LIN {X 0,Y 354.85,Z 275.906,A -85,B 0,C 180,E1 -13291.619,E2 -13291.619} C_VEL
LIN {X 0,Y 354.902,Z 275.901,A -85,B 0,C 180,E1 -13294.172,E2 -13294.172} C_VEL
LIN {X 0,Y 354.819,Z 275.911,A -85,B 0,C 180,E1 -13297.893,E2 -13297.893} C_VEL
LIN {X 0,Y 354.926,Z 275.898,A -85,B 0,C 180,E1 -13301.891,E2 -13301.891} C_VEL
LIN {X 0,Y 354.947,Z 275.897,A -85,B 0,C 180,E1 -13305.981,E2 -13305.981} C_VEL
LIN {X 0,Y 354.96,Z 275.894,A -85,B 0,C 180,E1 -13309.735,E2 -13309.735} C_VEL
LIN {X 0,Y 355.092,Z 275.876,A -85,B 0,C 180,E1 -13313.18,E2 -13313.18} C_VEL
LIN {X 0,Y 355.245,Z 275.86,A -85,B 0,C 180,E1 -13317.732,E2 -13317.732} C_VEL
LIN {X 0,Y 355.335,Z 275.85,A -85,B 0,C 180,E1 -13320,E2 -13320} C_VEL
LIN {X 0,Y 355.247,Z 275.86,A -85,B 0,C 180,E1 -13322.267,E2 -13322.267} C_VEL
LIN {X 0,Y 355.094,Z 275.875,A -85,B 0,C 180,E1 -13326.82,E2 -13326.82} C_VEL
LIN {X 0,Y 354.959,Z 275.894,A -85,B 0,C 180,E1 -13330.264,E2 -13330.264} C_VEL
LIN {X 0,Y 354.946,Z 275.896,A -85,B 0,C 180,E1 -13334.019,E2 -13334.019} C_VEL
LIN {X 0,Y 354.925,Z 275.898,A -85,B 0,C 180,E1 -13338.108,E2 -13338.108} C_VEL
LIN {X 0,Y 354.838,Z 275.908,A -85,B 0,C 180,E1 -13342.106,E2 -13342.106} C_VEL
LIN {X 0,Y 354.818,Z 275.914,A -85,B 0,C 180,E1 -13345.834,E2 -13345.834} C_VEL
LIN {X 0,Y 354.801,Z 275.915,A -85,B 0,C 180,E1 -13349.683,E2 -13349.683} C_VEL
LIN {X 0,Y 354.839,Z 276.09,A -85,B 0,C 180,E1 -13353.341,E2 -13353.341} C_VEL
LIN {X 0,Y 355.541,Z 279.989,A -85,B 0,C 180,E1 -13356.371,E2 -13356.371} C_VEL
LIN {X 0,Y 356.339,Z 284.55,A -85,B 0,C 180,E1 -13359.718,E2 -13359.718} C_VEL
LIN {X 0,Y 357.294,Z 289.71,A -85,B 0,C 180,E1 -13363.298,E2 -13363.298} C_VEL
LIN {X 0,Y 358.168,Z 294.793,A -85,B 0,C 180,E1 -13366.624,E2 -13366.624} C_VEL
LIN {X 0,Y 358.136,Z 298.563,A -85,B 0,C 180,E1 -13368.921,E2 -13368.921} C_VEL
LIN {X 0,Y 357.403,Z 304.661,A -85,B 0,C 180,E1 -13372.44,E2 -13372.44} C_VEL
LIN {X 0,Y 356.642,Z 310.823,A -85,B 0,C 180,E1 -13375.858,E2 -13375.858} C_VEL
LIN {X 0,Y 356.03,Z 316.866,A -85,B 0,C 180,E1 -13379.12,E2 -13379.12} C_VEL
LIN {X 0,Y 355.687,Z 320.46,A -85,B 0,C 180,E1 -13381.016,E2 -13381.016} C_VEL
LIN {X 0,Y 360.379,Z 339.057,A -85,B 0,C 180,E1 -13382.073,E2 -13382.073} C_VEL
LIN {X 0,Y 364.004,Z 355.046,A -85,B 0,C 180,E1 -13383.174,E2 -13383.174} C_VEL
LIN {X 0,Y 366.56,Z 369.171,A -85,B 0,C 180,E1 -13384.306,E2 -13384.306} C_VEL
LIN {X 0,Y 365.083,Z 383.132,A -85,B 0,C 180,E1 -13385.399,E2 -13385.399} C_VEL
LIN {X 0,Y 363.151,Z 396.131,A -85,B 0,C 180,E1 -13386.626,E2 -13386.626} C_VEL
LIN {X 0,Y 361.269,Z 409.429,A -85,B 0,C 180,E1 -13388.158,E2 -13388.158} C_VEL
LIN {X 0,Y 359.427,Z 421.341,A -85,B 0,C 180,E1 -13389.811,E2 -13389.811} C_VEL
LIN {X 0,Y 357.811,Z 432.557,A -85,B 0,C 180,E1 -13391.683,E2 -13391.683} C_VEL
LIN {X 0,Y 356.322,Z 442.487,A -85,B 0,C 180,E1 -13393.676,E2 -13393.676} C_VEL
LIN {X 0,Y 355.142,Z 451.425,A -85,B 0,C 180,E1 -13395.853,E2 -13395.853} C_VEL
LIN {X 0,Y 354.348,Z 458.565,A -85,B 0,C 180,E1 -13397.98,E2 -13397.98} C_VEL
LIN {X 0,Y 353.731,Z 464.736,A -85,B 0,C 180,E1 -13400.277,E2 -13400.277} C_VEL
LIN {X 0,Y 353.438,Z 469.47,A -85,B 0,C 180,E1 -13402.574,E2 -13402.574} C_VEL
LIN {X 0,Y 353.328,Z 472.143,A -85,B 0,C 180,E1 -13404.292,E2 -13404.292} C_VEL
LIN {X 0,Y 353.244,Z 474.612,A -85,B 0,C 180,E1 -13406.578,E2 -13406.578} C_VEL
LIN {X 0,Y 353.391,Z 475.823,A -85,B 0,C 180,E1 -13408.86,E2 -13408.86} C_VEL
LIN {X 0,Y 353.375,Z 475.789,A -85,B 0,C 180,E1 -13411.14,E2 -13411.14} C_VEL
LIN {X 0,Y 353.255,Z 474.542,A -85,B 0,C 180,E1 -13413.422,E2 -13413.422} C_VEL
LIN {X 0,Y 353.341,Z 472.092,A -85,B 0,C 180,E1 -13415.708,E2 -13415.708} C_VEL
LIN {X 0,Y 353.507,Z 468.395,A -85,B 0,C 180,E1 -13418,E2 -13418} C_VEL
LIN {X 0,Y 353.816,Z 463.389,A -85,B 0,C 180,E1 -13420.298,E2 -13420.298} C_VEL
LIN {X 0,Y 354.518,Z 456.97,A -85,B 0,C 180,E1 -13422.595,E2 -13422.595} C_VEL
LIN {X 0,Y 355.527,Z 449.023,A -85,B 0,C 180,E1 -13424.891,E2 -13424.891} C_VEL
LIN {X 0,Y 356.96,Z 439.375,A -85,B 0,C 180,E1 -13427.177,E2 -13427.177} C_VEL
LIN {X 0,Y 358.613,Z 429.339,A -85,B 0,C 180,E1 -13429.163,E2 -13429.163} C_VEL
LIN {X 0,Y 360.3,Z 419.297,A -85,B 0,C 180,E1 -13430.854,E2 -13430.854} C_VEL
LIN {X 0,Y 362.734,Z 405.658,A -85,B 0,C 180,E1 -13432.799,E2 -13432.799} C_VEL
LIN {X 0,Y 365.271,Z 391.753,A -85,B 0,C 180,E1 -13434.436,E2 -13434.436} C_VEL
LIN {X 0,Y 367.862,Z 377.541,A -85,B 0,C 180,E1 -13435.822,E2 -13435.822} C_VEL
LIN {X 0,Y 368.776,Z 371.059,A -85,B 0,C 180,E1 -13436.401,E2 -13436.401} C_VEL
LIN {X 0,Y 367.343,Z 351.718,A -85,B 0,C 180,E1 -13438.35,E2 -13438.35} C_VEL
LIN {X 0,Y 365.877,Z 341.967,A -85,B 0,C 180,E1 -13439.357,E2 -13439.357} C_VEL
LIN {X 0,Y 363.489,Z 331.98,A -85,B 0,C 180,E1 -13440.491,E2 -13440.491} C_VEL
LIN {X 0,Y 360.327,Z 322.118,A -85,B 0,C 180,E1 -13441.778,E2 -13441.778} C_VEL
LIN {X 0,Y 358.806,Z 317.901,A -85,B 0,C 180,E1 -13442.393,E2 -13442.393} C_VEL
LIN {X 0,Y 356.659,Z 312.833,A -85,B 0,C 180,E1 -13443.248,E2 -13443.248} C_VEL
LIN {X 0,Y 356.363,Z 310.972,A -85,B 0,C 180,E1 -13443.518,E2 -13443.518} C_VEL
LIN {X 0,Y 357.047,Z 306.93,A -85,B 0,C 180,E1 -13446.194,E2 -13446.194} C_VEL
LIN {X 0,Y 357.722,Z 303.241,A -85,B 0,C 180,E1 -13448.954,E2 -13448.954} C_VEL
LIN {X 0,Y 358.386,Z 299.982,A -85,B 0,C 180,E1 -13451.825,E2 -13451.825} C_VEL
LIN {X 0,Y 358.515,Z 298.431,A -85,B 0,C 180,E1 -13453.505,E2 -13453.505} C_VEL
LIN {X 0,Y 358.44,Z 297.199,A -85,B 0,C 180,E1 -13455.101,E2 -13455.101} C_VEL
LIN {X 0,Y 358.232,Z 296.25,A -85,B 0,C 180,E1 -13456.635,E2 -13456.635} C_VEL
LIN {X 0,Y 357.483,Z 294.847,A -85,B 0,C 180,E1 -13460.061,E2 -13460.061} C_VEL
LIN {X 0,Y 356.838,Z 294.398,A -85,B 0,C 180,E1 -13463.108,E2 -13463.108} C_VEL
LIN {X 0,Y 357.907,Z 296.935,A -85,B 0,C 180,E1 -13463.62,E2 -13463.62} C_VEL
LIN {X 0,Y 360.271,Z 300.003,A -85,B 0,C 180,E1 -13464.475,E2 -13464.475} C_VEL
LIN {X 0,Y 364.618,Z 306.868,A -85,B 0,C 180,E1 -13465.979,E2 -13465.979} C_VEL
LIN {X 0,Y 369.433,Z 316.686,A -85,B 0,C 180,E1 -13467.686,E2 -13467.686} C_VEL
LIN {X 0,Y 372.523,Z 325.556,A -85,B 0,C 180,E1 -13468.961,E2 -13468.961} C_VEL
LIN {X 0,Y 372.708,Z 327.732,A -85,B 0,C 180,E1 -13469.187,E2 -13469.187} C_VEL
LIN {X 0,Y 370.521,Z 341.272,A -85,B 0,C 180,E1 -13470.296,E2 -13470.296} C_VEL
LIN {X 0,Y 368.081,Z 355.561,A -85,B 0,C 180,E1 -13471.706,E2 -13471.706} C_VEL
LIN {X 0,Y 365.485,Z 369.993,A -85,B 0,C 180,E1 -13473.444,E2 -13473.444} C_VEL
LIN {X 0,Y 363.155,Z 382.14,A -85,B 0,C 180,E1 -13475.211,E2 -13475.211} C_VEL
LIN {X 0,Y 361.133,Z 392.946,A -85,B 0,C 180,E1 -13477.094,E2 -13477.094} C_VEL
LIN {X 0,Y 358.991,Z 403.616,A -85,B 0,C 180,E1 -13479.367,E2 -13479.367} C_VEL
LIN {X 0,Y 357.704,Z 410.335,A -85,B 0,C 180,E1 -13481.084,E2 -13481.084} C_VEL
LIN {X 0,Y 356.334,Z 417.681,A -85,B 0,C 180,E1 -13483.383,E2 -13483.383} C_VEL
LIN {X 0,Y 355.285,Z 423.605,A -85,B 0,C 180,E1 -13485.764,E2 -13485.764} C_VEL
LIN {X 0,Y 354.732,Z 426.779,A -85,B 0,C 180,E1 -13487.413,E2 -13487.413} C_VEL
LIN {X 0,Y 354.107,Z 430.099,A -85,B 0,C 180,E1 -13489.711,E2 -13489.711} C_VEL
LIN {X 0,Y 353.786,Z 432.114,A -85,B 0,C 180,E1 -13492.007,E2 -13492.007} C_VEL
LIN {X 0,Y 353.631,Z 432.891,A -85,B 0,C 180,E1 -13494.297,E2 -13494.297} C_VEL
LIN {X 0,Y 353.541,Z 432.443,A -85,B 0,C 180,E1 -13496.581,E2 -13496.581} C_VEL
LIN {X 0,Y 353.533,Z 430.76,A -85,B 0,C 180,E1 -13498.861,E2 -13498.861} C_VEL
LIN {X 0,Y 353.572,Z 427.813,A -85,B 0,C 180,E1 -13501.139,E2 -13501.139} C_VEL
LIN {X 0,Y 353.949,Z 423.542,A -85,B 0,C 180,E1 -13503.415,E2 -13503.415} C_VEL
LIN {X 0,Y 354.362,Z 419.416,A -85,B 0,C 180,E1 -13505.121,E2 -13505.121} C_VEL
LIN {X 0,Y 354.772,Z 412.637,A -85,B 0,C 180,E1 -13507.398,E2 -13507.398} C_VEL
LIN {X 0,Y 355.642,Z 404.164,A -85,B 0,C 180,E1 -13509.67,E2 -13509.67} C_VEL
LIN {X 0,Y 356.697,Z 395.156,A -85,B 0,C 180,E1 -13511.652,E2 -13511.652} C_VEL
LIN {X 0,Y 357.892,Z 384.378,A -85,B 0,C 180,E1 -13513.63,E2 -13513.63} C_VEL
LIN {X 0,Y 359.228,Z 373.388,A -85,B 0,C 180,E1 -13515.315,E2 -13515.315} C_VEL
LIN {X 0,Y 360.681,Z 360.339,A -85,B 0,C 180,E1 -13516.995,E2 -13516.995} C_VEL
LIN {X 0,Y 362.03,Z 347.331,A -85,B 0,C 180,E1 -13518.389,E2 -13518.389} C_VEL
LIN {X 0,Y 363.53,Z 333.259,A -85,B 0,C 180,E1 -13519.628,E2 -13519.628} C_VEL
LIN {X 0,Y 364.782,Z 317.486,A -85,B 0,C 180,E1 -13520.757,E2 -13520.757} C_VEL
LIN {X 0,Y 360.614,Z 301.762,A -85,B 0,C 180,E1 -13521.924,E2 -13521.924} C_VEL
LIN {X 0,Y 355.886,Z 285.872,A -85,B 0,C 180,E1 -13522.918,E2 -13522.918} C_VEL
LIN {X 0,Y 353.92,Z 279.21,A -85,B 0,C 180,E1 -13523.289,E2 -13523.289} C_VEL
LIN {X 0,Y 353.968,Z 276.176,A -85,B 0,C 180,E1 -13526.687,E2 -13526.687} C_VEL
LIN {X 0,Y 354.293,Z 275.978,A -85,B 0,C 180,E1 -13529.731,E2 -13529.731} C_VEL
LIN {X 0,Y 354.529,Z 275.947,A -85,B 0,C 180,E1 -13532.36,E2 -13532.36} C_VEL
LIN {X 0,Y 354.794,Z 275.914,A -85,B 0,C 180,E1 -13535.692,E2 -13535.692} C_VEL
LIN {X 0,Y 354.827,Z 275.912,A -85,B 0,C 180,E1 -13539.424,E2 -13539.424} C_VEL
LIN {X 0,Y 354.791,Z 275.918,A -85,B 0,C 180,E1 -13542.867,E2 -13542.867} C_VEL
LIN {X 0,Y 354.77,Z 275.916,A -85,B 0,C 180,E1 -13546.104,E2 -13546.104} C_VEL
LIN {X 0,Y 354.791,Z 275.916,A -85,B 0,C 180,E1 -13549.179,E2 -13549.179} C_VEL
LIN {X 0,Y 354.81,Z 275.913,A -85,B 0,C 180,E1 -13552.403,E2 -13552.403} C_VEL
LIN {X 0,Y 354.815,Z 275.914,A -85,B 0,C 180,E1 -13554.941,E2 -13554.941} C_VEL
LIN {X 0,Y 354.796,Z 275.916,A -85,B 0,C 180,E1 -13558.405,E2 -13558.405} C_VEL
LIN {X 0,Y 354.849,Z 275.906,A -85,B 0,C 180,E1 -13561.619,E2 -13561.619} C_VEL
LIN {X 0,Y 354.901,Z 275.902,A -85,B 0,C 180,E1 -13564.173,E2 -13564.173} C_VEL
LIN {X 0,Y 354.811,Z 275.912,A -85,B 0,C 180,E1 -13567.892,E2 -13567.892} C_VEL
LIN {X 0,Y 354.925,Z 275.898,A -85,B 0,C 180,E1 -13571.892,E2 -13571.892} C_VEL
LIN {X 0,Y 354.946,Z 275.897,A -85,B 0,C 180,E1 -13575.981,E2 -13575.981} C_VEL
LIN {X 0,Y 354.981,Z 275.891,A -85,B 0,C 180,E1 -13579.736,E2 -13579.736} C_VEL
LIN {X 0,Y 355.091,Z 275.876,A -85,B 0,C 180,E1 -13583.18,E2 -13583.18} C_VEL
LIN {X 0,Y 355.238,Z 275.861,A -85,B 0,C 180,E1 -13587.732,E2 -13587.732} C_VEL
LIN {X 0,Y 355.355,Z 275.848,A -85,B 0,C 180,E1 -13590,E2 -13590} C_VEL
LIN {X 0,Y 355.244,Z 275.859,A -85,B 0,C 180,E1 -13592.268,E2 -13592.268} C_VEL
LIN {X 0,Y 355.102,Z 275.875,A -85,B 0,C 180,E1 -13596.82,E2 -13596.82} C_VEL
LIN {X 0,Y 354.959,Z 275.894,A -85,B 0,C 180,E1 -13600.265,E2 -13600.265} C_VEL
LIN {X 0,Y 354.946,Z 275.896,A -85,B 0,C 180,E1 -13604.019,E2 -13604.019} C_VEL
LIN {X 0,Y 354.926,Z 275.898,A -85,B 0,C 180,E1 -13608.108,E2 -13608.108} C_VEL
LIN {X 0,Y 354.838,Z 275.908,A -85,B 0,C 180,E1 -13612.106,E2 -13612.106} C_VEL
LIN {X 0,Y 354.903,Z 275.902,A -85,B 0,C 180,E1 -13615.827,E2 -13615.827} C_VEL
LIN {X 0,Y 354.821,Z 275.912,A -85,B 0,C 180,E1 -13619.682,E2 -13619.682} C_VEL
LIN {X 0,Y 354.809,Z 275.913,A -85,B 0,C 180,E1 -13623.702,E2 -13623.702} C_VEL
LIN {X 0,Y 354.799,Z 275.912,A -85,B 0,C 180,E1 -13626.46,E2 -13626.46} C_VEL
LIN {X 0,Y 354.771,Z 275.919,A -85,B 0,C 180,E1 -13629.412,E2 -13629.412} C_VEL
LIN {X 0,Y 354.787,Z 275.918,A -85,B 0,C 180,E1 -13632.866,E2 -13632.866} C_VEL
LIN {X 0,Y 354.769,Z 275.916,A -85,B 0,C 180,E1 -13636.104,E2 -13636.104} C_VEL
LIN {X 0,Y 354.785,Z 275.917,A -85,B 0,C 180,E1 -13638.708,E2 -13638.708} C_VEL
LIN {X 0,Y 354.146,Z 276.003,A -85,B 0,C 180,E1 -13639.657,E2 -13639.657} C_VEL
LIN {X 0,Y 351.276,Z 276.358,A -85,B 0,C 180,E1 -13641.199,E2 -13641.199} C_VEL
LIN {X 0,Y 348.845,Z 276.656,A -85,B 0,C 180,E1 -13642.447,E2 -13642.447} C_VEL
LIN {X 0,Y 347.829,Z 276.781,A -85,B 0,C 180,E1 -13643.413,E2 -13643.413} C_VEL
LIN {X 0,Y 347.762,Z 276.788,A -85,B 0,C 180,E1 -13643.741,E2 -13643.741} C_VEL
LIN {X 0,Y 347.737,Z 276.796,A -85,B 0,C 180,E1 -13646.928,E2 -13646.928} C_VEL
LIN {X 0,Y 347.782,Z 276.789,A -85,B 0,C 180,E1 -13650.988,E2 -13650.988} C_VEL
LIN {X 0,Y 347.834,Z 276.779,A -85,B 0,C 180,E1 -13653.608,E2 -13653.608} C_VEL
LIN {X 0,Y 347.789,Z 276.788,A -85,B 0,C 180,E1 -13656.162,E2 -13656.162} C_VEL
LIN {X 0,Y 347.811,Z 276.784,A -85,B 0,C 180,E1 -13659.909,E2 -13659.909} C_VEL
LIN {X 0,Y 347.87,Z 276.78,A -85,B 0,C 180,E1 -13662.359,E2 -13662.359} C_VEL
LIN {X 0,Y 347.901,Z 276.774,A -85,B 0,C 180,E1 -13665.971,E2 -13665.971} C_VEL
LIN {X 0,Y 347.901,Z 276.772,A -85,B 0,C 180,E1 -13669.524,E2 -13669.524} C_VEL
LIN {X 0,Y 348.059,Z 276.752,A -85,B 0,C 180,E1 -13673.041,E2 -13673.041} C_VEL
LIN {X 0,Y 348.207,Z 276.736,A -85,B 0,C 180,E1 -13677.686,E2 -13677.686} C_VEL
LIN {X 0,Y 348.287,Z 276.728,A -85,B 0,C 180,E1 -13680,E2 -13680} C_VEL
LIN {X 0,Y 348.21,Z 276.736,A -85,B 0,C 180,E1 -13682.313,E2 -13682.313} C_VEL
LIN {X 0,Y 348.06,Z 276.751,A -85,B 0,C 180,E1 -13686.958,E2 -13686.958} C_VEL
LIN {X 0,Y 347.9,Z 276.772,A -85,B 0,C 180,E1 -13690.475,E2 -13690.475} C_VEL
LIN {X 0,Y 347.902,Z 276.773,A -85,B 0,C 180,E1 -13694.149,E2 -13694.149} C_VEL
LIN {X 0,Y 347.894,Z 276.773,A -85,B 0,C 180,E1 -13698.29,E2 -13698.29} C_VEL
LIN {X 0,Y 347.793,Z 276.789,A -85,B 0,C 180,E1 -13701.635,E2 -13701.635} C_VEL
LIN {X 0,Y 347.772,Z 276.79,A -85,B 0,C 180,E1 -13705.111,E2 -13705.111} C_VEL
LIN {X 0,Y 347.738,Z 276.794,A -85,B 0,C 180,E1 -13707.7,E2 -13707.7} C_VEL
LIN {X 0,Y 347.742,Z 276.794,A -85,B 0,C 180,E1 -13710.348,E2 -13710.348} C_VEL
LIN {X 0,Y 347.759,Z 276.839,A -85,B 0,C 180,E1 -13712.752,E2 -13712.752} C_VEL
LIN {X 0,Y 348.553,Z 281.23,A -85,B 0,C 180,E1 -13716.241,E2 -13716.241} C_VEL
LIN {X 0,Y 349.482,Z 286.512,A -85,B 0,C 180,E1 -13720.166,E2 -13720.166} C_VEL
LIN {X 0,Y 350.247,Z 290.566,A -85,B 0,C 180,E1 -13723.018,E2 -13723.018} C_VEL
LIN {X 0,Y 351.056,Z 295.188,A -85,B 0,C 180,E1 -13726.113,E2 -13726.113} C_VEL
LIN {X 0,Y 351.239,Z 297.774,A -85,B 0,C 180,E1 -13727.76,E2 -13727.76} C_VEL
LIN {X 0,Y 350.724,Z 302.912,A -85,B 0,C 180,E1 -13730.834,E2 -13730.834} C_VEL
LIN {X 0,Y 349.923,Z 309.065,A -85,B 0,C 180,E1 -13734.377,E2 -13734.377} C_VEL
LIN {X 0,Y 349.265,Z 315.014,A -85,B 0,C 180,E1 -13737.686,E2 -13737.686} C_VEL
LIN {X 0,Y 348.706,Z 320.201,A -85,B 0,C 180,E1 -13740.492,E2 -13740.492} C_VEL
LIN {X 0,Y 353.123,Z 337.808,A -85,B 0,C 180,E1 -13741.507,E2 -13741.507} C_VEL
LIN {X 0,Y 356.956,Z 354.401,A -85,B 0,C 180,E1 -13742.679,E2 -13742.679} C_VEL
LIN {X 0,Y 359.766,Z 370.145,A -85,B 0,C 180,E1 -13743.975,E2 -13743.975} C_VEL
LIN {X 0,Y 359.333,Z 375.801,A -85,B 0,C 180,E1 -13744.416,E2 -13744.416} C_VEL
LIN {X 0,Y 357.43,Z 389.485,A -85,B 0,C 180,E1 -13745.612,E2 -13745.612} C_VEL
LIN {X 0,Y 355.468,Z 402.63,A -85,B 0,C 180,E1 -13747.015,E2 -13747.015} C_VEL
LIN {X 0,Y 353.448,Z 415.792,A -85,B 0,C 180,E1 -13748.722,E2 -13748.722} C_VEL
LIN {X 0,Y 351.707,Z 426.828,A -85,B 0,C 180,E1 -13750.445,E2 -13750.445} C_VEL
LIN {X 0,Y 350.016,Z 437.641,A -85,B 0,C 180,E1 -13752.471,E2 -13752.471} C_VEL
LIN {X 0,Y 348.709,Z 446.678,A -85,B 0,C 180,E1 -13754.511,E2 -13754.511} C_VEL
LIN {X 0,Y 347.757,Z 454.196,A -85,B 0,C 180,E1 -13756.561,E2 -13756.561} C_VEL
LIN {X 0,Y 346.976,Z 461.209,A -85,B 0,C 180,E1 -13758.906,E2 -13758.906} C_VEL
LIN {X 0,Y 346.496,Z 466.696,A -85,B 0,C 180,E1 -13761.25,E2 -13761.25} C_VEL
LIN {X 0,Y 346.314,Z 469.901,A -85,B 0,C 180,E1 -13763.006,E2 -13763.006} C_VEL
LIN {X 0,Y 346.218,Z 473.045,A -85,B 0,C 180,E1 -13765.343,E2 -13765.343} C_VEL
LIN {X 0,Y 346.201,Z 474.903,A -85,B 0,C 180,E1 -13767.673,E2 -13767.673} C_VEL
LIN {X 0,Y 346.311,Z 475.366,A -85,B 0,C 180,E1 -13768.837,E2 -13768.837} C_VEL
LIN {X 0,Y 346.297,Z 475.367,A -85,B 0,C 180,E1 -13771.163,E2 -13771.163} C_VEL
LIN {X 0,Y 346.176,Z 474.151,A -85,B 0,C 180,E1 -13773.492,E2 -13773.492} C_VEL
LIN {X 0,Y 346.285,Z 471.458,A -85,B 0,C 180,E1 -13776.028,E2 -13776.028} C_VEL
LIN {X 0,Y 346.427,Z 468.077,A -85,B 0,C 180,E1 -13778.164,E2 -13778.164} C_VEL
LIN {X 0,Y 346.767,Z 463.108,A -85,B 0,C 180,E1 -13780.51,E2 -13780.51} C_VEL
LIN {X 0,Y 347.506,Z 456.739,A -85,B 0,C 180,E1 -13782.854,E2 -13782.854} C_VEL
LIN {X 0,Y 348.59,Z 448.878,A -85,B 0,C 180,E1 -13785.195,E2 -13785.195} C_VEL
LIN {X 0,Y 350.118,Z 439.372,A -85,B 0,C 180,E1 -13787.524,E2 -13787.524} C_VEL
LIN {X 0,Y 351.864,Z 429.469,A -85,B 0,C 180,E1 -13789.546,E2 -13789.546} C_VEL
LIN {X 0,Y 353.998,Z 417.872,A -85,B 0,C 180,E1 -13791.548,E2 -13791.548} C_VEL
LIN {X 0,Y 356.631,Z 404.158,A -85,B 0,C 180,E1 -13793.52,E2 -13793.52} C_VEL
LIN {X 0,Y 359.38,Z 390.278,A -85,B 0,C 180,E1 -13795.172,E2 -13795.172} C_VEL
LIN {X 0,Y 362.3,Z 375.244,A -85,B 0,C 180,E1 -13796.653,E2 -13796.653} C_VEL
LIN {X 0,Y 362.592,Z 372.475,A -85,B 0,C 180,E1 -13796.925,E2 -13796.925} C_VEL
LIN {X 0,Y 361.547,Z 353.176,A -85,B 0,C 180,E1 -13798.986,E2 -13798.986} C_VEL
LIN {X 0,Y 359.907,Z 342.138,A -85,B 0,C 180,E1 -13800.231,E2 -13800.231} C_VEL
LIN {X 0,Y 357.553,Z 332.291,A -85,B 0,C 180,E1 -13801.489,E2 -13801.489} C_VEL
LIN {X 0,Y 356.069,Z 327.128,A -85,B 0,C 180,E1 -13802.203,E2 -13802.203} C_VEL
LIN {X 0,Y 354.474,Z 322.345,A -85,B 0,C 180,E1 -13802.949,E2 -13802.949} C_VEL
LIN {X 0,Y 352.61,Z 317.64,A -85,B 0,C 180,E1 -13803.79,E2 -13803.79} C_VEL
LIN {X 0,Y 352.385,Z 316.525,A -85,B 0,C 180,E1 -13803.948,E2 -13803.948} C_VEL
LIN {X 0,Y 350.293,Z 311.942,A -85,B 0,C 180,E1 -13804.934,E2 -13804.934} C_VEL
LIN {X 0,Y 349.808,Z 309.463,A -85,B 0,C 180,E1 -13805.353,E2 -13805.353} C_VEL
LIN {X 0,Y 350.649,Z 305.114,A -85,B 0,C 180,E1 -13808.587,E2 -13808.587} C_VEL
LIN {X 0,Y 351.322,Z 302.003,A -85,B 0,C 180,E1 -13811.311,E2 -13811.311} C_VEL
LIN {X 0,Y 351.565,Z 299.578,A -85,B 0,C 180,E1 -13813.974,E2 -13813.974} C_VEL
LIN {X 0,Y 351.37,Z 298.141,A -85,B 0,C 180,E1 -13816.06,E2 -13816.06} C_VEL
LIN {X 0,Y 350.861,Z 296.886,A -85,B 0,C 180,E1 -13818.623,E2 -13818.623} C_VEL
LIN {X 0,Y 350.289,Z 296.173,A -85,B 0,C 180,E1 -13821.282,E2 -13821.282} C_VEL
LIN {X 0,Y 350.697,Z 297.494,A -85,B 0,C 180,E1 -13821.593,E2 -13821.593} C_VEL
LIN {X 0,Y 351.72,Z 299.107,A -85,B 0,C 180,E1 -13822.118,E2 -13822.118} C_VEL
LIN {X 0,Y 353.274,Z 300.437,A -85,B 0,C 180,E1 -13822.727,E2 -13822.727} C_VEL
LIN {X 0,Y 355.163,Z 303.662,A -85,B 0,C 180,E1 -13823.584,E2 -13823.584} C_VEL
LIN {X 0,Y 358.458,Z 308.693,A -85,B 0,C 180,E1 -13824.883,E2 -13824.883} C_VEL
LIN {X 0,Y 362.509,Z 316.531,A -85,B 0,C 180,E1 -13826.476,E2 -13826.476} C_VEL
LIN {X 0,Y 365.589,Z 324.049,A -85,B 0,C 180,E1 -13827.763,E2 -13827.763} C_VEL
LIN {X 0,Y 367.18,Z 329.285,A -85,B 0,C 180,E1 -13828.535,E2 -13828.535} C_VEL
LIN {X 0,Y 364.385,Z 345.126,A -85,B 0,C 180,E1 -13829.903,E2 -13829.903} C_VEL
LIN {X 0,Y 361.806,Z 358.925,A -85,B 0,C 180,E1 -13831.362,E2 -13831.362} C_VEL
LIN {X 0,Y 359.307,Z 371.574,A -85,B 0,C 180,E1 -13832.95,E2 -13832.95} C_VEL
LIN {X 0,Y 356.579,Z 384.833,A -85,B 0,C 180,E1 -13834.97,E2 -13834.97} C_VEL
LIN {X 0,Y 354.351,Z 395.455,A -85,B 0,C 180,E1 -13836.939,E2 -13836.939} C_VEL
LIN {X 0,Y 352.393,Z 404.582,A -85,B 0,C 180,E1 -13838.962,E2 -13838.962} C_VEL
LIN {X 0,Y 350.595,Z 413.15,A -85,B 0,C 180,E1 -13841.293,E2 -13841.293} C_VEL
LIN {X 0,Y 349.202,Z 420.004,A -85,B 0,C 180,E1 -13843.635,E2 -13843.635} C_VEL
LIN {X 0,Y 348.214,Z 425.335,A -85,B 0,C 180,E1 -13845.984,E2 -13845.984} C_VEL
LIN {X 0,Y 347.341,Z 429.262,A -85,B 0,C 180,E1 -13848.327,E2 -13848.327} C_VEL
LIN {X 0,Y 346.899,Z 431.859,A -85,B 0,C 180,E1 -13850.673,E2 -13850.673} C_VEL
LIN {X 0,Y 346.609,Z 433.214,A -85,B 0,C 180,E1 -13853.012,E2 -13853.012} C_VEL
LIN {X 0,Y 346.454,Z 433.33,A -85,B 0,C 180,E1 -13855.346,E2 -13855.346} C_VEL
LIN {X 0,Y 346.509,Z 432.212,A -85,B 0,C 180,E1 -13857.675,E2 -13857.675} C_VEL
LIN {X 0,Y 346.447,Z 429.864,A -85,B 0,C 180,E1 -13860,E2 -13860} C_VEL
LIN {X 0,Y 346.669,Z 426.21,A -85,B 0,C 180,E1 -13862.324,E2 -13862.324} C_VEL
LIN {X 0,Y 347.157,Z 421.199,A -85,B 0,C 180,E1 -13864.645,E2 -13864.645} C_VEL
LIN {X 0,Y 347.601,Z 414.75,A -85,B 0,C 180,E1 -13866.968,E2 -13866.968} C_VEL
LIN {X 0,Y 348.375,Z 406.661,A -85,B 0,C 180,E1 -13869.288,E2 -13869.288} C_VEL
LIN {X 0,Y 349.39,Z 398.055,A -85,B 0,C 180,E1 -13871.311,E2 -13871.311} C_VEL
LIN {X 0,Y 350.619,Z 387.75,A -85,B 0,C 180,E1 -13873.328,E2 -13873.328} C_VEL
LIN {X 0,Y 351.866,Z 377.299,A -85,B 0,C 180,E1 -13875.05,E2 -13875.05} C_VEL
LIN {X 0,Y 353.381,Z 364.902,A -85,B 0,C 180,E1 -13876.761,E2 -13876.761} C_VEL
LIN {X 0,Y 354.824,Z 351.082,A -85,B 0,C 180,E1 -13878.35,E2 -13878.35} C_VEL
LIN {X 0,Y 356.276,Z 337.965,A -85,B 0,C 180,E1 -13879.594,E2 -13879.594} C_VEL
LIN {X 0,Y 357.575,Z 323.561,A -85,B 0,C 180,E1 -13880.719,E2 -13880.719} C_VEL
LIN {X 0,Y 357.86,Z 318.505,A -85,B 0,C 180,E1 -13881.07,E2 -13881.07} C_VEL
LIN {X 0,Y 353.728,Z 302.534,A -85,B 0,C 180,E1 -13882.293,E2 -13882.293} C_VEL
LIN {X 0,Y 348.767,Z 286.075,A -85,B 0,C 180,E1 -13883.345,E2 -13883.345} C_VEL
LIN {X 0,Y 346.865,Z 279.6,A -85,B 0,C 180,E1 -13883.739,E2 -13883.739} C_VEL
LIN {X 0,Y 346.916,Z 276.901,A -85,B 0,C 180,E1 -13886.953,E2 -13886.953} C_VEL
LIN {X 0,Y 347.302,Z 276.846,A -85,B 0,C 180,E1 -13890.392,E2 -13890.392} C_VEL
LIN {X 0,Y 347.646,Z 276.803,A -85,B 0,C 180,E1 -13894.018,E2 -13894.018} C_VEL
LIN {X 0,Y 347.758,Z 276.793,A -85,B 0,C 180,E1 -13897.322,E2 -13897.322} C_VEL
LIN {X 0,Y 347.734,Z 276.793,A -85,B 0,C 180,E1 -13900.297,E2 -13900.297} C_VEL
LIN {X 0,Y 347.726,Z 276.795,A -85,B 0,C 180,E1 -13903.408,E2 -13903.408} C_VEL
LIN {X 0,Y 347.728,Z 276.797,A -85,B 0,C 180,E1 -13906.686,E2 -13906.686} C_VEL
LIN {X 0,Y 347.75,Z 276.791,A -85,B 0,C 180,E1 -13910.173,E2 -13910.173} C_VEL
LIN {X 0,Y 347.764,Z 276.793,A -85,B 0,C 180,E1 -13912.679,E2 -13912.679} C_VEL
LIN {X 0,Y 347.751,Z 276.79,A -85,B 0,C 180,E1 -13915.956,E2 -13915.956} C_VEL
LIN {X 0,Y 347.752,Z 276.79,A -85,B 0,C 180,E1 -13919.652,E2 -13919.652} C_VEL
LIN {X 0,Y 347.833,Z 276.78,A -85,B 0,C 180,E1 -13923.608,E2 -13923.608} C_VEL
LIN {X 0,Y 347.785,Z 276.789,A -85,B 0,C 180,E1 -13926.161,E2 -13926.161} C_VEL
LIN {X 0,Y 347.81,Z 276.784,A -85,B 0,C 180,E1 -13929.909,E2 -13929.909} C_VEL
LIN {X 0,Y 347.869,Z 276.78,A -85,B 0,C 180,E1 -13932.359,E2 -13932.359} C_VEL
LIN {X 0,Y 347.901,Z 276.775,A -85,B 0,C 180,E1 -13935.971,E2 -13935.971} C_VEL
LIN {X 0,Y 347.931,Z 276.768,A -85,B 0,C 180,E1 -13939.526,E2 -13939.526} C_VEL
LIN {X 0,Y 348.058,Z 276.752,A -85,B 0,C 180,E1 -13943.041,E2 -13943.041} C_VEL
LIN {X 0,Y 348.199,Z 276.737,A -85,B 0,C 180,E1 -13947.686,E2 -13947.686} C_VEL
LIN {X 0,Y 348.306,Z 276.726,A -85,B 0,C 180,E1 -13950,E2 -13950} C_VEL
LIN {X 0,Y 348.206,Z 276.735,A -85,B 0,C 180,E1 -13952.314,E2 -13952.314} C_VEL
LIN {X 0,Y 348.067,Z 276.751,A -85,B 0,C 180,E1 -13956.959,E2 -13956.959} C_VEL
LIN {X 0,Y 347.899,Z 276.772,A -85,B 0,C 180,E1 -13960.475,E2 -13960.475} C_VEL
LIN {X 0,Y 347.902,Z 276.773,A -85,B 0,C 180,E1 -13964.15,E2 -13964.15} C_VEL
LIN {X 0,Y 347.894,Z 276.773,A -85,B 0,C 180,E1 -13968.29,E2 -13968.29} C_VEL
LIN {X 0,Y 347.792,Z 276.789,A -85,B 0,C 180,E1 -13971.635,E2 -13971.635} C_VEL
LIN {X 0,Y 347.816,Z 276.785,A -85,B 0,C 180,E1 -13975.108,E2 -13975.108} C_VEL
LIN {X 0,Y 347.811,Z 276.785,A -85,B 0,C 180,E1 -13977.694,E2 -13977.694} C_VEL
LIN {X 0,Y 347.752,Z 276.79,A -85,B 0,C 180,E1 -13980.348,E2 -13980.348} C_VEL
LIN {X 0,Y 347.751,Z 276.79,A -85,B 0,C 180,E1 -13984.044,E2 -13984.044} C_VEL
LIN {X 0,Y 347.759,Z 276.793,A -85,B 0,C 180,E1 -13987.321,E2 -13987.321} C_VEL
LIN {X 0,Y 347.744,Z 276.792,A -85,B 0,C 180,E1 -13991.601,E2 -13991.601} C_VEL
LIN {X 0,Y 347.707,Z 276.8,A -85,B 0,C 180,E1 -13995.027,E2 -13995.027} C_VEL
LIN {X 0,Y 347.734,Z 276.791,A -85,B 0,C 180,E1 -13998.699,E2 -13998.699} C_VEL
LIN {X 0,Y 347.777,Z 276.787,A -85,B 0,C 180,E1 -14002.011,E2 -14002.011} C_VEL
LIN {X 0,Y 347.762,Z 276.788,A -85,B 0,C 180,E1 -14003.741,E2 -14003.741} C_VEL
LIN {X 0,Y 347.122,Z 276.873,A -85,B 0,C 180,E1 -14004.706,E2 -14004.706} C_VEL
LIN {X 0,Y 344.232,Z 277.23,A -85,B 0,C 180,E1 -14006.276,E2 -14006.276} C_VEL
LIN {X 0,Y 341.782,Z 277.533,A -85,B 0,C 180,E1 -14007.547,E2 -14007.547} C_VEL
LIN {X 0,Y 340.761,Z 277.665,A -85,B 0,C 180,E1 -14008.531,E2 -14008.531} C_VEL
LIN {X 0,Y 340.696,Z 277.671,A -85,B 0,C 180,E1 -14008.865,E2 -14008.865} C_VEL
LIN {X 0,Y 340.78,Z 277.663,A -85,B 0,C 180,E1 -14012.475,E2 -14012.475} C_VEL
LIN {X 0,Y 340.758,Z 277.661,A -85,B 0,C 180,E1 -14015.638,E2 -14015.638} C_VEL
LIN {X 0,Y 340.738,Z 277.663,A -85,B 0,C 180,E1 -14019.473,E2 -14019.473} C_VEL
LIN {X 0,Y 340.862,Z 277.65,A -85,B 0,C 180,E1 -14021.984,E2 -14021.984} C_VEL
LIN {X 0,Y 340.873,Z 277.648,A -85,B 0,C 180,E1 -14025.705,E2 -14025.705} C_VEL
LIN {X 0,Y 340.852,Z 277.649,A -85,B 0,C 180,E1 -14029.305,E2 -14029.305} C_VEL
LIN {X 0,Y 341.006,Z 277.63,A -85,B 0,C 180,E1 -14032.896,E2 -14032.896} C_VEL
LIN {X 0,Y 341.168,Z 277.612,A -85,B 0,C 180,E1 -14037.638,E2 -14037.638} C_VEL
LIN {X 0,Y 341.239,Z 277.606,A -85,B 0,C 180,E1 -14040,E2 -14040} C_VEL
LIN {X 0,Y 341.171,Z 277.612,A -85,B 0,C 180,E1 -14042.361,E2 -14042.361} C_VEL
LIN {X 0,Y 341.007,Z 277.63,A -85,B 0,C 180,E1 -14047.103,E2 -14047.103} C_VEL
LIN {X 0,Y 340.851,Z 277.649,A -85,B 0,C 180,E1 -14050.694,E2 -14050.694} C_VEL
LIN {X 0,Y 340.866,Z 277.648,A -85,B 0,C 180,E1 -14054.324,E2 -14054.324} C_VEL
LIN {X 0,Y 340.84,Z 277.651,A -85,B 0,C 180,E1 -14058.466,E2 -14058.466} C_VEL
LIN {X 0,Y 340.756,Z 277.664,A -85,B 0,C 180,E1 -14061.856,E2 -14061.856} C_VEL
LIN {X 0,Y 340.723,Z 277.67,A -85,B 0,C 180,E1 -14065.668,E2 -14065.668} C_VEL
LIN {X 0,Y 340.71,Z 277.671,A -85,B 0,C 180,E1 -14069.673,E2 -14069.673} C_VEL
LIN {X 0,Y 340.76,Z 277.881,A -85,B 0,C 180,E1 -14072.428,E2 -14072.428} C_VEL
LIN {X 0,Y 341.345,Z 281.303,A -85,B 0,C 180,E1 -14075.204,E2 -14075.204} C_VEL
LIN {X 0,Y 342.141,Z 285.823,A -85,B 0,C 180,E1 -14078.687,E2 -14078.687} C_VEL
LIN {X 0,Y 343.14,Z 291.103,A -85,B 0,C 180,E1 -14082.523,E2 -14082.523} C_VEL
LIN {X 0,Y 344.034,Z 296.202,A -85,B 0,C 180,E1 -14086.007,E2 -14086.007} C_VEL
LIN {X 0,Y 344.245,Z 298.724,A -85,B 0,C 180,E1 -14087.645,E2 -14087.645} C_VEL
LIN {X 0,Y 343.739,Z 303.659,A -85,B 0,C 180,E1 -14090.667,E2 -14090.667} C_VEL
LIN {X 0,Y 342.906,Z 309.789,A -85,B 0,C 180,E1 -14094.259,E2 -14094.259} C_VEL
LIN {X 0,Y 342.188,Z 315.883,A -85,B 0,C 180,E1 -14097.724,E2 -14097.724} C_VEL
LIN {X 0,Y 341.752,Z 319.867,A -85,B 0,C 180,E1 -14099.938,E2 -14099.938} C_VEL
LIN {X 0,Y 346.223,Z 337.818,A -85,B 0,C 180,E1 -14101.016,E2 -14101.016} C_VEL
LIN {X 0,Y 349.775,Z 353.361,A -85,B 0,C 180,E1 -14102.139,E2 -14102.139} C_VEL
LIN {X 0,Y 352.635,Z 368.759,A -85,B 0,C 180,E1 -14103.428,E2 -14103.428} C_VEL
LIN {X 0,Y 352.977,Z 373.292,A -85,B 0,C 180,E1 -14103.831,E2 -14103.831} C_VEL
LIN {X 0,Y 351.132,Z 386.693,A -85,B 0,C 180,E1 -14104.987,E2 -14104.987} C_VEL
LIN {X 0,Y 349.181,Z 398.96,A -85,B 0,C 180,E1 -14106.263,E2 -14106.263} C_VEL
LIN {X 0,Y 347.186,Z 411.6,A -85,B 0,C 180,E1 -14107.851,E2 -14107.851} C_VEL
LIN {X 0,Y 345.186,Z 424.094,A -85,B 0,C 180,E1 -14109.75,E2 -14109.75} C_VEL
LIN {X 0,Y 343.665,Z 433.825,A -85,B 0,C 180,E1 -14111.52,E2 -14111.52} C_VEL
LIN {X 0,Y 342.124,Z 443.405,A -85,B 0,C 180,E1 -14113.593,E2 -14113.593} C_VEL
LIN {X 0,Y 340.9,Z 451.97,A -85,B 0,C 180,E1 -14115.841,E2 -14115.841} C_VEL
LIN {X 0,Y 340.115,Z 458.912,A -85,B 0,C 180,E1 -14118.075,E2 -14118.075} C_VEL
LIN {X 0,Y 339.509,Z 464.832,A -85,B 0,C 180,E1 -14120.468,E2 -14120.468} C_VEL
LIN {X 0,Y 339.24,Z 469.347,A -85,B 0,C 180,E1 -14122.859,E2 -14122.859} C_VEL
LIN {X 0,Y 339.136,Z 472.535,A -85,B 0,C 180,E1 -14125.245,E2 -14125.245} C_VEL
LIN {X 0,Y 339.111,Z 474.416,A -85,B 0,C 180,E1 -14127.624,E2 -14127.624} C_VEL
LIN {X 0,Y 339.233,Z 474.901,A -85,B 0,C 180,E1 -14128.813,E2 -14128.813} C_VEL
LIN {X 0,Y 339.204,Z 474.942,A -85,B 0,C 180,E1 -14131.187,E2 -14131.187} C_VEL
LIN {X 0,Y 339.1,Z 473.766,A -85,B 0,C 180,E1 -14133.565,E2 -14133.565} C_VEL
LIN {X 0,Y 339.205,Z 471.312,A -85,B 0,C 180,E1 -14136.007,E2 -14136.007} C_VEL
LIN {X 0,Y 339.364,Z 467.778,A -85,B 0,C 180,E1 -14138.335,E2 -14138.335} C_VEL
LIN {X 0,Y 339.729,Z 462.845,A -85,B 0,C 180,E1 -14140.73,E2 -14140.73} C_VEL
LIN {X 0,Y 340.511,Z 456.55,A -85,B 0,C 180,E1 -14143.123,E2 -14143.123} C_VEL
LIN {X 0,Y 341.653,Z 448.786,A -85,B 0,C 180,E1 -14145.511,E2 -14145.511} C_VEL
LIN {X 0,Y 343.284,Z 439.412,A -85,B 0,C 180,E1 -14147.884,E2 -14147.884} C_VEL
LIN {X 0,Y 345.145,Z 429.679,A -85,B 0,C 180,E1 -14149.942,E2 -14149.942} C_VEL
LIN {X 0,Y 347.415,Z 418.307,A -85,B 0,C 180,E1 -14151.978,E2 -14151.978} C_VEL
LIN {X 0,Y 350.192,Z 404.983,A -85,B 0,C 180,E1 -14153.979,E2 -14153.979} C_VEL
LIN {X 0,Y 353.332,Z 390.297,A -85,B 0,C 180,E1 -14155.792,E2 -14155.792} C_VEL
LIN {X 0,Y 356.406,Z 375.629,A -85,B 0,C 180,E1 -14157.289,E2 -14157.289} C_VEL
LIN {X 0,Y 355.93,Z 355.427,A -85,B 0,C 180,E1 -14159.58,E2 -14159.58} C_VEL
LIN {X 0,Y 354.516,Z 344.772,A -85,B 0,C 180,E1 -14160.868,E2 -14160.868} C_VEL
LIN {X 0,Y 352.423,Z 335.168,A -85,B 0,C 180,E1 -14162.192,E2 -14162.192} C_VEL
LIN {X 0,Y 350.246,Z 327.385,A -85,B 0,C 180,E1 -14163.424,E2 -14163.424} C_VEL
LIN {X 0,Y 348.082,Z 320.862,A -85,B 0,C 180,E1 -14164.636,E2 -14164.636} C_VEL
LIN {X 0,Y 346.682,Z 317.378,A -85,B 0,C 180,E1 -14165.412,E2 -14165.412} C_VEL
LIN {X 0,Y 346.297,Z 315.645,A -85,B 0,C 180,E1 -14165.729,E2 -14165.729} C_VEL
LIN {X 0,Y 344.024,Z 310.449,A -85,B 0,C 180,E1 -14167.182,E2 -14167.182} C_VEL
LIN {X 0,Y 343.442,Z 307.426,A -85,B 0,C 180,E1 -14167.872,E2 -14167.872} C_VEL
LIN {X 0,Y 344.299,Z 303.861,A -85,B 0,C 180,E1 -14170.952,E2 -14170.952} C_VEL
LIN {X 0,Y 344.597,Z 302.118,A -85,B 0,C 180,E1 -14172.759,E2 -14172.759} C_VEL
LIN {X 0,Y 344.626,Z 300.752,A -85,B 0,C 180,E1 -14174.459,E2 -14174.459} C_VEL
LIN {X 0,Y 344.216,Z 299.028,A -85,B 0,C 180,E1 -14177.31,E2 -14177.31} C_VEL
LIN {X 0,Y 343.927,Z 298.47,A -85,B 0,C 180,E1 -14178.842,E2 -14178.842} C_VEL
LIN {X 0,Y 344.998,Z 300.803,A -85,B 0,C 180,E1 -14179.81,E2 -14179.81} C_VEL
LIN {X 0,Y 347.364,Z 303.167,A -85,B 0,C 180,E1 -14181.156,E2 -14181.156} C_VEL
LIN {X 0,Y 348.552,Z 305.244,A -85,B 0,C 180,E1 -14181.848,E2 -14181.848} C_VEL
LIN {X 0,Y 349.524,Z 306.13,A -85,B 0,C 180,E1 -14182.269,E2 -14182.269} C_VEL
LIN {X 0,Y 354.172,Z 313.76,A -85,B 0,C 180,E1 -14184.448,E2 -14184.448} C_VEL
LIN {X 0,Y 357.121,Z 319.607,A -85,B 0,C 180,E1 -14185.746,E2 -14185.746} C_VEL
LIN {X 0,Y 360.37,Z 327.697,A -85,B 0,C 180,E1 -14187.25,E2 -14187.25} C_VEL
LIN {X 0,Y 361.511,Z 332.446,A -85,B 0,C 180,E1 -14187.983,E2 -14187.983} C_VEL
LIN {X 0,Y 358.845,Z 346.301,A -85,B 0,C 180,E1 -14189.226,E2 -14189.226} C_VEL
LIN {X 0,Y 355.752,Z 361.526,A -85,B 0,C 180,E1 -14190.891,E2 -14190.891} C_VEL
LIN {X 0,Y 353.201,Z 373.281,A -85,B 0,C 180,E1 -14192.443,E2 -14192.443} C_VEL
LIN {X 0,Y 350.616,Z 384.745,A -85,B 0,C 180,E1 -14194.227,E2 -14194.227} C_VEL
LIN {X 0,Y 348.24,Z 395.276,A -85,B 0,C 180,E1 -14196.195,E2 -14196.195} C_VEL
LIN {X 0,Y 346.127,Z 404.433,A -85,B 0,C 180,E1 -14198.25,E2 -14198.25} C_VEL
LIN {X 0,Y 344.335,Z 412.149,A -85,B 0,C 180,E1 -14200.32,E2 -14200.32} C_VEL
LIN {X 0,Y 342.754,Z 419.286,A -85,B 0,C 180,E1 -14202.704,E2 -14202.704} C_VEL
LIN {X 0,Y 341.779,Z 423.639,A -85,B 0,C 180,E1 -14204.495,E2 -14204.495} C_VEL
LIN {X 0,Y 340.873,Z 428.158,A -85,B 0,C 180,E1 -14206.892,E2 -14206.892} C_VEL
LIN {X 0,Y 340.072,Z 431.369,A -85,B 0,C 180,E1 -14209.281,E2 -14209.281} C_VEL
LIN {X 0,Y 339.69,Z 433.276,A -85,B 0,C 180,E1 -14211.673,E2 -14211.673} C_VEL
LIN {X 0,Y 339.491,Z 433.954,A -85,B 0,C 180,E1 -14214.059,E2 -14214.059} C_VEL
LIN {X 0,Y 339.361,Z 433.405,A -85,B 0,C 180,E1 -14216.438,E2 -14216.438} C_VEL
LIN {X 0,Y 339.407,Z 431.616,A -85,B 0,C 180,E1 -14218.814,E2 -14218.814} C_VEL
LIN {X 0,Y 339.446,Z 428.582,A -85,B 0,C 180,E1 -14221.187,E2 -14221.187} C_VEL
LIN {X 0,Y 339.792,Z 424.21,A -85,B 0,C 180,E1 -14223.558,E2 -14223.558} C_VEL
LIN {X 0,Y 340.222,Z 419.972,A -85,B 0,C 180,E1 -14225.334,E2 -14225.334} C_VEL
LIN {X 0,Y 340.722,Z 412.819,A -85,B 0,C 180,E1 -14227.779,E2 -14227.779} C_VEL
LIN {X 0,Y 341.641,Z 404.441,A -85,B 0,C 180,E1 -14230.071,E2 -14230.071} C_VEL
LIN {X 0,Y 342.793,Z 395.288,A -85,B 0,C 180,E1 -14232.131,E2 -14232.131} C_VEL
LIN {X 0,Y 344.058,Z 384.352,A -85,B 0,C 180,E1 -14234.189,E2 -14234.189} C_VEL
LIN {X 0,Y 345.617,Z 372.208,A -85,B 0,C 180,E1 -14236.085,E2 -14236.085} C_VEL
LIN {X 0,Y 347.067,Z 359.972,A -85,B 0,C 180,E1 -14237.683,E2 -14237.683} C_VEL
LIN {X 0,Y 348.55,Z 346.774,A -85,B 0,C 180,E1 -14239.127,E2 -14239.127} C_VEL
LIN {X 0,Y 350.117,Z 332.473,A -85,B 0,C 180,E1 -14240.413,E2 -14240.413} C_VEL
LIN {X 0,Y 350.963,Z 319.388,A -85,B 0,C 180,E1 -14241.394,E2 -14241.394} C_VEL
LIN {X 0,Y 347.129,Z 304.659,A -85,B 0,C 180,E1 -14242.559,E2 -14242.559} C_VEL
LIN {X 0,Y 342.342,Z 288.399,A -85,B 0,C 180,E1 -14243.656,E2 -14243.656} C_VEL
LIN {X 0,Y 339.814,Z 279.975,A -85,B 0,C 180,E1 -14244.165,E2 -14244.165} C_VEL
LIN {X 0,Y 339.902,Z 277.774,A -85,B 0,C 180,E1 -14247.058,E2 -14247.058} C_VEL
LIN {X 0,Y 340.207,Z 277.731,A -85,B 0,C 180,E1 -14249.814,E2 -14249.814} C_VEL
LIN {X 0,Y 340.451,Z 277.7,A -85,B 0,C 180,E1 -14252.461,E2 -14252.461} C_VEL
LIN {X 0,Y 340.671,Z 277.676,A -85,B 0,C 180,E1 -14255.285,E2 -14255.285} C_VEL
LIN {X 0,Y 340.711,Z 277.667,A -85,B 0,C 180,E1 -14258.386,E2 -14258.386} C_VEL
LIN {X 0,Y 340.701,Z 277.668,A -85,B 0,C 180,E1 -14262.045,E2 -14262.045} C_VEL
LIN {X 0,Y 340.655,Z 277.674,A -85,B 0,C 180,E1 -14266.227,E2 -14266.227} C_VEL
LIN {X 0,Y 340.691,Z 277.669,A -85,B 0,C 180,E1 -14269.753,E2 -14269.753} C_VEL
LIN {X 0,Y 340.708,Z 277.669,A -85,B 0,C 180,E1 -14273.258,E2 -14273.258} C_VEL
LIN {X 0,Y 340.695,Z 277.67,A -85,B 0,C 180,E1 -14276.153,E2 -14276.153} C_VEL
LIN {X 0,Y 340.744,Z 277.666,A -85,B 0,C 180,E1 -14280.329,E2 -14280.329} C_VEL
LIN {X 0,Y 340.806,Z 277.657,A -85,B 0,C 180,E1 -14283.02,E2 -14283.02} C_VEL
LIN {X 0,Y 340.756,Z 277.661,A -85,B 0,C 180,E1 -14285.638,E2 -14285.638} C_VEL
LIN {X 0,Y 340.737,Z 277.664,A -85,B 0,C 180,E1 -14289.473,E2 -14289.473} C_VEL
LIN {X 0,Y 340.861,Z 277.65,A -85,B 0,C 180,E1 -14291.984,E2 -14291.984} C_VEL
LIN {X 0,Y 340.872,Z 277.648,A -85,B 0,C 180,E1 -14295.705,E2 -14295.705} C_VEL
LIN {X 0,Y 340.874,Z 277.647,A -85,B 0,C 180,E1 -14299.306,E2 -14299.306} C_VEL
LIN {X 0,Y 341.005,Z 277.631,A -85,B 0,C 180,E1 -14302.897,E2 -14302.897} C_VEL
LIN {X 0,Y 340.829,Z 277.652,A -85,B 0,C 180,E1 -14305.269,E2 -14305.269} C_VEL
LIN {X 0,Y 341.16,Z 277.613,A -85,B 0,C 180,E1 -14307.639,E2 -14307.639} C_VEL
LIN {X 0,Y 341.257,Z 277.604,A -85,B 0,C 180,E1 -14310,E2 -14310} C_VEL
LIN {X 0,Y 341.167,Z 277.612,A -85,B 0,C 180,E1 -14312.361,E2 -14312.361} C_VEL
LIN {X 0,Y 341.012,Z 277.63,A -85,B 0,C 180,E1 -14317.103,E2 -14317.103} C_VEL
LIN {X 0,Y 340.851,Z 277.649,A -85,B 0,C 180,E1 -14320.695,E2 -14320.695} C_VEL
LIN {X 0,Y 340.866,Z 277.648,A -85,B 0,C 180,E1 -14324.325,E2 -14324.325} C_VEL
LIN {X 0,Y 340.84,Z 277.651,A -85,B 0,C 180,E1 -14328.466,E2 -14328.466} C_VEL
LIN {X 0,Y 340.757,Z 277.663,A -85,B 0,C 180,E1 -14331.857,E2 -14331.857} C_VEL
LIN {X 0,Y 340.776,Z 277.662,A -85,B 0,C 180,E1 -14335.664,E2 -14335.664} C_VEL
LIN {X 0,Y 340.732,Z 277.664,A -85,B 0,C 180,E1 -14338.321,E2 -14338.321} C_VEL
LIN {X 0,Y 340.701,Z 277.671,A -85,B 0,C 180,E1 -14341.045,E2 -14341.045} C_VEL
LIN {X 0,Y 340.721,Z 277.671,A -85,B 0,C 180,E1 -14345.279,E2 -14345.279} C_VEL
LIN {X 0,Y 340.696,Z 277.669,A -85,B 0,C 180,E1 -14348.383,E2 -14348.383} C_VEL
LIN {X 0,Y 340.696,Z 277.669,A -85,B 0,C 180,E1 -14352.044,E2 -14352.044} C_VEL
LIN {X 0,Y 340.655,Z 277.674,A -85,B 0,C 180,E1 -14356.227,E2 -14356.227} C_VEL
LIN {X 0,Y 340.692,Z 277.669,A -85,B 0,C 180,E1 -14359.753,E2 -14359.753} C_VEL
LIN {X 0,Y 340.708,Z 277.669,A -85,B 0,C 180,E1 -14363.258,E2 -14363.258} C_VEL
LIN {X 0,Y 340.696,Z 277.67,A -85,B 0,C 180,E1 -14366.153,E2 -14366.153} C_VEL
LIN {X 0,Y 340.696,Z 277.671,A -85,B 0,C 180,E1 -14368.865,E2 -14368.865} C_VEL
LIN {X 0,Y 340.085,Z 277.754,A -85,B 0,C 180,E1 -14369.852,E2 -14369.852} C_VEL
LIN {X 0,Y 337.28,Z 278.103,A -85,B 0,C 180,E1 -14371.46,E2 -14371.46} C_VEL
LIN {X 0,Y 334.864,Z 278.399,A -85,B 0,C 180,E1 -14372.762,E2 -14372.762} C_VEL
LIN {X 0,Y 333.811,Z 278.526,A -85,B 0,C 180,E1 -14373.769,E2 -14373.769} C_VEL
LIN {X 0,Y 333.719,Z 278.537,A -85,B 0,C 180,E1 -14374.11,E2 -14374.11} C_VEL
LIN {X 0,Y 333.668,Z 278.545,A -85,B 0,C 180,E1 -14377.937,E2 -14377.937} C_VEL
LIN {X 0,Y 333.798,Z 278.528,A -85,B 0,C 180,E1 -14381.589,E2 -14381.589} C_VEL
LIN {X 0,Y 333.812,Z 278.526,A -85,B 0,C 180,E1 -14385.576,E2 -14385.576} C_VEL
LIN {X 0,Y 333.822,Z 278.525,A -85,B 0,C 180,E1 -14389.077,E2 -14389.077} C_VEL
LIN {X 0,Y 333.961,Z 278.509,A -85,B 0,C 180,E1 -14392.746,E2 -14392.746} C_VEL
LIN {X 0,Y 333.796,Z 278.528,A -85,B 0,C 180,E1 -14395.169,E2 -14395.169} C_VEL
LIN {X 0,Y 334.105,Z 278.491,A -85,B 0,C 180,E1 -14397.589,E2 -14397.589} C_VEL
LIN {X 0,Y 334.191,Z 278.484,A -85,B 0,C 180,E1 -14400,E2 -14400} C_VEL
LIN {X 0,Y 334.109,Z 278.491,A -85,B 0,C 180,E1 -14402.411,E2 -14402.411} C_VEL
LIN {X 0,Y 333.996,Z 278.507,A -85,B 0,C 180,E1 -14406.039,E2 -14406.039} C_VEL
LIN {X 0,Y 333.824,Z 278.529,A -85,B 0,C 180,E1 -14409.696,E2 -14409.696} C_VEL
LIN {X 0,Y 333.8,Z 278.53,A -85,B 0,C 180,E1 -14413.391,E2 -14413.391} C_VEL
LIN {X 0,Y 333.75,Z 278.535,A -85,B 0,C 180,E1 -14417.146,E2 -14417.146} C_VEL
LIN {X 0,Y 333.742,Z 278.54,A -85,B 0,C 180,E1 -14419.69,E2 -14419.69} C_VEL
LIN {X 0,Y 333.694,Z 278.541,A -85,B 0,C 180,E1 -14422.278,E2 -14422.278} C_VEL
LIN {X 0,Y 333.692,Z 278.543,A -85,B 0,C 180,E1 -14425.09,E2 -14425.09} C_VEL
LIN {X 0,Y 333.656,Z 278.549,A -85,B 0,C 180,E1 -14428.977,E2 -14428.977} C_VEL
LIN {X 0,Y 333.643,Z 278.564,A -85,B 0,C 180,E1 -14431.777,E2 -14431.777} C_VEL
LIN {X 0,Y 334.321,Z 282.341,A -85,B 0,C 180,E1 -14434.93,E2 -14434.93} C_VEL
LIN {X 0,Y 335.223,Z 287.509,A -85,B 0,C 180,E1 -14438.973,E2 -14438.973} C_VEL
LIN {X 0,Y 336.042,Z 291.609,A -85,B 0,C 180,E1 -14442.009,E2 -14442.009} C_VEL
LIN {X 0,Y 336.825,Z 296.142,A -85,B 0,C 180,E1 -14445.188,E2 -14445.188} C_VEL
LIN {X 0,Y 337.227,Z 299.638,A -85,B 0,C 180,E1 -14447.523,E2 -14447.523} C_VEL
LIN {X 0,Y 336.734,Z 304.494,A -85,B 0,C 180,E1 -14450.554,E2 -14450.554} C_VEL
LIN {X 0,Y 335.883,Z 310.473,A -85,B 0,C 180,E1 -14454.135,E2 -14454.135} C_VEL
LIN {X 0,Y 335.152,Z 316.566,A -85,B 0,C 180,E1 -14457.674,E2 -14457.674} C_VEL
LIN {X 0,Y 334.787,Z 319.63,A -85,B 0,C 180,E1 -14459.394,E2 -14459.394} C_VEL
LIN {X 0,Y 339.072,Z 336.904,A -85,B 0,C 180,E1 -14460.453,E2 -14460.453} C_VEL
LIN {X 0,Y 342.778,Z 353.202,A -85,B 0,C 180,E1 -14461.655,E2 -14461.655} C_VEL
LIN {X 0,Y 345.692,Z 368.925,A -85,B 0,C 180,E1 -14463.015,E2 -14463.015} C_VEL
LIN {X 0,Y 346.243,Z 373.867,A -85,B 0,C 180,E1 -14463.477,E2 -14463.477} C_VEL
LIN {X 0,Y 344.382,Z 386.756,A -85,B 0,C 180,E1 -14464.624,E2 -14464.624} C_VEL
LIN {X 0,Y 342.227,Z 400.163,A -85,B 0,C 180,E1 -14466.072,E2 -14466.072} C_VEL
LIN {X 0,Y 340.169,Z 412.525,A -85,B 0,C 180,E1 -14467.689,E2 -14467.689} C_VEL
LIN {X 0,Y 338.153,Z 424.801,A -85,B 0,C 180,E1 -14469.627,E2 -14469.627} C_VEL
LIN {X 0,Y 336.576,Z 434.348,A -85,B 0,C 180,E1 -14471.432,E2 -14471.432} C_VEL
LIN {X 0,Y 335.031,Z 443.773,A -85,B 0,C 180,E1 -14473.549,E2 -14473.549} C_VEL
LIN {X 0,Y 333.985,Z 450.917,A -85,B 0,C 180,E1 -14475.459,E2 -14475.459} C_VEL
LIN {X 0,Y 333.103,Z 458.202,A -85,B 0,C 180,E1 -14477.82,E2 -14477.82} C_VEL
LIN {X 0,Y 332.447,Z 464.188,A -85,B 0,C 180,E1 -14480.263,E2 -14480.263} C_VEL
LIN {X 0,Y 332.165,Z 468.764,A -85,B 0,C 180,E1 -14482.707,E2 -14482.707} C_VEL
LIN {X 0,Y 332.059,Z 471.987,A -85,B 0,C 180,E1 -14485.143,E2 -14485.143} C_VEL
LIN {X 0,Y 332.022,Z 473.917,A -85,B 0,C 180,E1 -14487.574,E2 -14487.574} C_VEL
LIN {X 0,Y 332.14,Z 474.426,A -85,B 0,C 180,E1 -14488.787,E2 -14488.787} C_VEL
LIN {X 0,Y 332.111,Z 474.515,A -85,B 0,C 180,E1 -14491.213,E2 -14491.213} C_VEL
LIN {X 0,Y 332.026,Z 473.39,A -85,B 0,C 180,E1 -14493.641,E2 -14493.641} C_VEL
LIN {X 0,Y 332.121,Z 471.066,A -85,B 0,C 180,E1 -14496.074,E2 -14496.074} C_VEL
LIN {X 0,Y 332.294,Z 467.482,A -85,B 0,C 180,E1 -14498.514,E2 -14498.514} C_VEL
LIN {X 0,Y 332.692,Z 462.612,A -85,B 0,C 180,E1 -14500.96,E2 -14500.96} C_VEL
LIN {X 0,Y 333.533,Z 456.402,A -85,B 0,C 180,E1 -14503.402,E2 -14503.402} C_VEL
LIN {X 0,Y 334.957,Z 447.72,A -85,B 0,C 180,E1 -14506.141,E2 -14506.141} C_VEL
LIN {X 0,Y 336.735,Z 438.292,A -85,B 0,C 180,E1 -14508.559,E2 -14508.559} C_VEL
LIN {X 0,Y 338.723,Z 428.525,A -85,B 0,C 180,E1 -14510.654,E2 -14510.654} C_VEL
LIN {X 0,Y 341.247,Z 417.156,A -85,B 0,C 180,E1 -14512.716,E2 -14512.716} C_VEL
LIN {X 0,Y 344.274,Z 403.882,A -85,B 0,C 180,E1 -14514.739,E2 -14514.739} C_VEL
LIN {X 0,Y 347.611,Z 389.326,A -85,B 0,C 180,E1 -14516.572,E2 -14516.572} C_VEL
LIN {X 0,Y 350.31,Z 377.685,A -85,B 0,C 180,E1 -14517.804,E2 -14517.804} C_VEL
LIN {X 0,Y 350.464,Z 362.63,A -85,B 0,C 180,E1 -14519.614,E2 -14519.614} C_VEL
LIN {X 0,Y 350.135,Z 354.492,A -85,B 0,C 180,E1 -14520.598,E2 -14520.598} C_VEL
LIN {X 0,Y 348.526,Z 343.323,A -85,B 0,C 180,E1 -14522.121,E2 -14522.121} C_VEL
LIN {X 0,Y 346.744,Z 335.17,A -85,B 0,C 180,E1 -14523.409,E2 -14523.409} C_VEL
LIN {X 0,Y 344.64,Z 327.594,A -85,B 0,C 180,E1 -14524.819,E2 -14524.819} C_VEL
LIN {X 0,Y 342.281,Z 319.875,A -85,B 0,C 180,E1 -14526.545,E2 -14526.545} C_VEL
LIN {X 0,Y 340.642,Z 315.206,A -85,B 0,C 180,E1 -14527.88,E2 -14527.88} C_VEL
LIN {X 0,Y 340.364,Z 313.416,A -85,B 0,C 180,E1 -14528.313,E2 -14528.313} C_VEL
LIN {X 0,Y 338.682,Z 309.671,A -85,B 0,C 180,E1 -14530.037,E2 -14530.037} C_VEL
LIN {X 0,Y 338.011,Z 306.237,A -85,B 0,C 180,E1 -14531.71,E2 -14531.71} C_VEL
LIN {X 0,Y 337.935,Z 304.887,A -85,B 0,C 180,E1 -14532.524,E2 -14532.524} C_VEL
LIN {X 0,Y 337.92,Z 304.034,A -85,B 0,C 180,E1 -14533.341,E2 -14533.341} C_VEL
LIN {X 0,Y 338.194,Z 303.516,A -85,B 0,C 180,E1 -14535.045,E2 -14535.045} C_VEL
LIN {X 0,Y 339.181,Z 304.206,A -85,B 0,C 180,E1 -14536.861,E2 -14536.861} C_VEL
LIN {X 0,Y 341.297,Z 305.451,A -85,B 0,C 180,E1 -14538.781,E2 -14538.781} C_VEL
LIN {X 0,Y 342.762,Z 307.809,A -85,B 0,C 180,E1 -14539.993,E2 -14539.993} C_VEL
LIN {X 0,Y 344.245,Z 309.323,A -85,B 0,C 180,E1 -14540.878,E2 -14540.878} C_VEL
LIN {X 0,Y 347.245,Z 314.125,A -85,B 0,C 180,E1 -14542.614,E2 -14542.614} C_VEL
LIN {X 0,Y 350.101,Z 319.086,A -85,B 0,C 180,E1 -14544.064,E2 -14544.064} C_VEL
LIN {X 0,Y 353.064,Z 325.617,A -85,B 0,C 180,E1 -14545.581,E2 -14545.581} C_VEL
LIN {X 0,Y 355.488,Z 332.397,A -85,B 0,C 180,E1 -14546.906,E2 -14546.906} C_VEL
LIN {X 0,Y 356.053,Z 334.57,A -85,B 0,C 180,E1 -14547.278,E2 -14547.278} C_VEL
LIN {X 0,Y 353.12,Z 349.046,A -85,B 0,C 180,E1 -14548.671,E2 -14548.671} C_VEL
LIN {X 0,Y 350.103,Z 362.596,A -85,B 0,C 180,E1 -14550.209,E2 -14550.209} C_VEL
LIN {X 0,Y 347.141,Z 375.131,A -85,B 0,C 180,E1 -14551.92,E2 -14551.92} C_VEL
LIN {X 0,Y 344.457,Z 386.034,A -85,B 0,C 180,E1 -14553.688,E2 -14553.688} C_VEL
LIN {X 0,Y 341.848,Z 396.565,A -85,B 0,C 180,E1 -14555.722,E2 -14555.722} C_VEL
LIN {X 0,Y 339.633,Z 405.577,A -85,B 0,C 180,E1 -14557.812,E2 -14557.812} C_VEL
LIN {X 0,Y 337.695,Z 413.119,A -85,B 0,C 180,E1 -14559.917,E2 -14559.917} C_VEL
LIN {X 0,Y 335.994,Z 420.166,A -85,B 0,C 180,E1 -14562.345,E2 -14562.345} C_VEL
LIN {X 0,Y 334.929,Z 424.444,A -85,B 0,C 180,E1 -14564.17,E2 -14564.17} C_VEL
LIN {X 0,Y 333.951,Z 428.901,A -85,B 0,C 180,E1 -14566.615,E2 -14566.615} C_VEL
LIN {X 0,Y 333.076,Z 432.02,A -85,B 0,C 180,E1 -14569.053,E2 -14569.053} C_VEL
LIN {X 0,Y 332.666,Z 433.876,A -85,B 0,C 180,E1 -14571.496,E2 -14571.496} C_VEL
LIN {X 0,Y 332.437,Z 434.49,A -85,B 0,C 180,E1 -14573.933,E2 -14573.933} C_VEL
LIN {X 0,Y 332.277,Z 433.88,A -85,B 0,C 180,E1 -14576.362,E2 -14576.362} C_VEL
LIN {X 0,Y 332.328,Z 432.032,A -85,B 0,C 180,E1 -14578.789,E2 -14578.789} C_VEL
LIN {X 0,Y 332.368,Z 428.928,A -85,B 0,C 180,E1 -14581.212,E2 -14581.212} C_VEL
LIN {X 0,Y 332.712,Z 424.496,A -85,B 0,C 180,E1 -14583.634,E2 -14583.634} C_VEL
LIN {X 0,Y 333.145,Z 420.219,A -85,B 0,C 180,E1 -14585.448,E2 -14585.448} C_VEL
LIN {X 0,Y 333.65,Z 413.532,A -85,B 0,C 180,E1 -14587.778,E2 -14587.778} C_VEL
LIN {X 0,Y 334.495,Z 405.732,A -85,B 0,C 180,E1 -14589.982,E2 -14589.982} C_VEL
LIN {X 0,Y 335.655,Z 396.724,A -85,B 0,C 180,E1 -14592.086,E2 -14592.086} C_VEL
LIN {X 0,Y 336.954,Z 385.955,A -85,B 0,C 180,E1 -14594.187,E2 -14594.187} C_VEL
LIN {X 0,Y 338.392,Z 375.001,A -85,B 0,C 180,E1 -14595.973,E2 -14595.973} C_VEL
LIN {X 0,Y 339.991,Z 362.018,A -85,B 0,C 180,E1 -14597.752,E2 -14597.752} C_VEL
LIN {X 0,Y 341.435,Z 349.123,A -85,B 0,C 180,E1 -14599.229,E2 -14599.229} C_VEL
LIN {X 0,Y 343.081,Z 335.252,A -85,B 0,C 180,E1 -14600.537,E2 -14600.537} C_VEL
LIN {X 0,Y 344.243,Z 321.189,A -85,B 0,C 180,E1 -14601.637,E2 -14601.637} C_VEL
LIN {X 0,Y 340.234,Z 305.721,A -85,B 0,C 180,E1 -14602.911,E2 -14602.911} C_VEL
LIN {X 0,Y 335.383,Z 289.158,A -85,B 0,C 180,E1 -14604.075,E2 -14604.075} C_VEL
LIN {X 0,Y 332.746,Z 280.335,A -85,B 0,C 180,E1 -14604.624,E2 -14604.624} C_VEL
LIN {X 0,Y 332.749,Z 278.871,A -85,B 0,C 180,E1 -14606.33,E2 -14606.33} C_VEL
LIN {X 0,Y 333.042,Z 278.627,A -85,B 0,C 180,E1 -14609.036,E2 -14609.036} C_VEL
LIN {X 0,Y 333.407,Z 278.577,A -85,B 0,C 180,E1 -14612.523,E2 -14612.523} C_VEL
LIN {X 0,Y 333.594,Z 278.555,A -85,B 0,C 180,E1 -14614.751,E2 -14614.751} C_VEL
LIN {X 0,Y 333.65,Z 278.547,A -85,B 0,C 180,E1 -14617.652,E2 -14617.652} C_VEL
LIN {X 0,Y 333.649,Z 278.55,A -85,B 0,C 180,E1 -14620.768,E2 -14620.768} C_VEL
LIN {X 0,Y 333.596,Z 278.553,A -85,B 0,C 180,E1 -14624.25,E2 -14624.25} C_VEL
LIN {X 0,Y 333.644,Z 278.547,A -85,B 0,C 180,E1 -14627.619,E2 -14627.619} C_VEL
LIN {X 0,Y 333.655,Z 278.548,A -85,B 0,C 180,E1 -14631.202,E2 -14631.202} C_VEL
LIN {X 0,Y 333.679,Z 278.543,A -85,B 0,C 180,E1 -14633.861,E2 -14633.861} C_VEL
LIN {X 0,Y 333.646,Z 278.547,A -85,B 0,C 180,E1 -14637.413,E2 -14637.413} C_VEL
LIN {X 0,Y 333.693,Z 278.543,A -85,B 0,C 180,E1 -14641.026,E2 -14641.026} C_VEL
LIN {X 0,Y 333.737,Z 278.536,A -85,B 0,C 180,E1 -14643.754,E2 -14643.754} C_VEL
LIN {X 0,Y 333.657,Z 278.546,A -85,B 0,C 180,E1 -14647.719,E2 -14647.719} C_VEL
LIN {X 0,Y 333.797,Z 278.528,A -85,B 0,C 180,E1 -14651.59,E2 -14651.59} C_VEL
LIN {X 0,Y 333.811,Z 278.527,A -85,B 0,C 180,E1 -14655.577,E2 -14655.577} C_VEL
LIN {X 0,Y 333.837,Z 278.523,A -85,B 0,C 180,E1 -14659.078,E2 -14659.078} C_VEL
LIN {X 0,Y 333.96,Z 278.508,A -85,B 0,C 180,E1 -14662.746,E2 -14662.746} C_VEL
LIN {X 0,Y 333.794,Z 278.528,A -85,B 0,C 180,E1 -14665.169,E2 -14665.169} C_VEL
LIN {X 0,Y 334.097,Z 278.493,A -85,B 0,C 180,E1 -14667.589,E2 -14667.589} C_VEL
LIN {X 0,Y 334.209,Z 278.482,A -85,B 0,C 180,E1 -14670,E2 -14670} C_VEL
LIN {X 0,Y 334.105,Z 278.491,A -85,B 0,C 180,E1 -14672.411,E2 -14672.411} C_VEL
LIN {X 0,Y 334,Z 278.506,A -85,B 0,C 180,E1 -14676.039,E2 -14676.039} C_VEL
LIN {X 0,Y 333.824,Z 278.53,A -85,B 0,C 180,E1 -14679.696,E2 -14679.696} C_VEL
LIN {X 0,Y 333.8,Z 278.531,A -85,B 0,C 180,E1 -14683.391,E2 -14683.391} C_VEL
LIN {X 0,Y 333.75,Z 278.536,A -85,B 0,C 180,E1 -14687.146,E2 -14687.146} C_VEL
LIN {X 0,Y 333.742,Z 278.539,A -85,B 0,C 180,E1 -14689.69,E2 -14689.69} C_VEL
LIN {X 0,Y 333.696,Z 278.541,A -85,B 0,C 180,E1 -14692.278,E2 -14692.278} C_VEL
LIN {X 0,Y 333.738,Z 278.535,A -85,B 0,C 180,E1 -14696.246,E2 -14696.246} C_VEL
LIN {X 0,Y 333.693,Z 278.543,A -85,B 0,C 180,E1 -14698.974,E2 -14698.974} C_VEL
LIN {X 0,Y 333.647,Z 278.547,A -85,B 0,C 180,E1 -14702.587,E2 -14702.587} C_VEL
LIN {X 0,Y 333.678,Z 278.543,A -85,B 0,C 180,E1 -14706.139,E2 -14706.139} C_VEL
LIN {X 0,Y 333.623,Z 278.555,A -85,B 0,C 180,E1 -14709.196,E2 -14709.196} C_VEL
LIN {X 0,Y 333.631,Z 278.55,A -85,B 0,C 180,E1 -14712.499,E2 -14712.499} C_VEL
LIN {X 0,Y 333.599,Z 278.553,A -85,B 0,C 180,E1 -14715.955,E2 -14715.955} C_VEL
LIN {X 0,Y 333.651,Z 278.548,A -85,B 0,C 180,E1 -14719.315,E2 -14719.315} C_VEL
LIN {X 0,Y 333.669,Z 278.546,A -85,B 0,C 180,E1 -14723.168,E2 -14723.168} C_VEL
LIN {X 0,Y 333.678,Z 278.544,A -85,B 0,C 180,E1 -14725.341,E2 -14725.341} C_VEL
LIN {X 0,Y 333.694,Z 278.541,A -85,B 0,C 180,E1 -14729.637,E2 -14729.637} C_VEL
LIN {X 0,Y 333.743,Z 278.538,A -85,B 0,C 180,E1 -14732.401,E2 -14732.401} C_VEL
LIN {X 0,Y 333.719,Z 278.537,A -85,B 0,C 180,E1 -14734.11,E2 -14734.11} C_VEL
LIN {X 0,Y 333.021,Z 278.627,A -85,B 0,C 180,E1 -14735.118,E2 -14735.118} C_VEL
LIN {X 0,Y 330.122,Z 278.989,A -85,B 0,C 180,E1 -14736.756,E2 -14736.756} C_VEL
LIN {X 0,Y 327.701,Z 279.289,A -85,B 0,C 180,E1 -14738.084,E2 -14738.084} C_VEL
LIN {X 0,Y 326.696,Z 279.414,A -85,B 0,C 180,E1 -14739.112,E2 -14739.112} C_VEL
LIN {X 0,Y 326.631,Z 279.42,A -85,B 0,C 180,E1 -14739.46,E2 -14739.46} C_VEL
LIN {X 0,Y 326.704,Z 279.416,A -85,B 0,C 180,E1 -14742.472,E2 -14742.472} C_VEL
LIN {X 0,Y 326.763,Z 279.41,A -85,B 0,C 180,E1 -14746.314,E2 -14746.314} C_VEL
LIN {X 0,Y 326.787,Z 279.405,A -85,B 0,C 180,E1 -14750.093,E2 -14750.093} C_VEL
LIN {X 0,Y 326.948,Z 279.384,A -85,B 0,C 180,E1 -14753.83,E2 -14753.83} C_VEL
LIN {X 0,Y 327.045,Z 279.37,A -85,B 0,C 180,E1 -14757.536,E2 -14757.536} C_VEL
LIN {X 0,Y 327.144,Z 279.362,A -85,B 0,C 180,E1 -14760,E2 -14760} C_VEL
LIN {X 0,Y 327.049,Z 279.37,A -85,B 0,C 180,E1 -14762.463,E2 -14762.463} C_VEL
LIN {X 0,Y 326.95,Z 279.384,A -85,B 0,C 180,E1 -14766.17,E2 -14766.17} C_VEL
LIN {X 0,Y 326.786,Z 279.406,A -85,B 0,C 180,E1 -14769.907,E2 -14769.907} C_VEL
LIN {X 0,Y 326.762,Z 279.41,A -85,B 0,C 180,E1 -14773.685,E2 -14773.685} C_VEL
LIN {X 0,Y 326.703,Z 279.416,A -85,B 0,C 180,E1 -14777.527,E2 -14777.527} C_VEL
LIN {X 0,Y 326.669,Z 279.417,A -85,B 0,C 180,E1 -14780.134,E2 -14780.134} C_VEL
LIN {X 0,Y 326.639,Z 279.42,A -85,B 0,C 180,E1 -14784.13,E2 -14784.13} C_VEL
LIN {X 0,Y 326.6,Z 279.426,A -85,B 0,C 180,E1 -14788.256,E2 -14788.256} C_VEL
LIN {X 0,Y 326.637,Z 279.596,A -85,B 0,C 180,E1 -14791.451,E2 -14791.451} C_VEL
LIN {X 0,Y 327.138,Z 282.539,A -85,B 0,C 180,E1 -14793.956,E2 -14793.956} C_VEL
LIN {X 0,Y 327.913,Z 286.944,A -85,B 0,C 180,E1 -14797.532,E2 -14797.532} C_VEL
LIN {X 0,Y 328.94,Z 292.27,A -85,B 0,C 180,E1 -14801.6,E2 -14801.6} C_VEL
LIN {X 0,Y 329.843,Z 297.464,A -85,B 0,C 180,E1 -14805.321,E2 -14805.321} C_VEL
LIN {X 0,Y 330.161,Z 300.029,A -85,B 0,C 180,E1 -14807.064,E2 -14807.064} C_VEL
LIN {X 0,Y 329.893,Z 303.729,A -85,B 0,C 180,E1 -14809.454,E2 -14809.454} C_VEL
LIN {X 0,Y 329.054,Z 309.908,A -85,B 0,C 180,E1 -14813.271,E2 -14813.271} C_VEL
LIN {X 0,Y 328.086,Z 317.215,A -85,B 0,C 180,E1 -14817.62,E2 -14817.62} C_VEL
LIN {X 0,Y 327.816,Z 319.28,A -85,B 0,C 180,E1 -14818.825,E2 -14818.825} C_VEL
LIN {X 0,Y 332.34,Z 337.911,A -85,B 0,C 180,E1 -14820.001,E2 -14820.001} C_VEL
LIN {X 0,Y 335.914,Z 353.909,A -85,B 0,C 180,E1 -14821.236,E2 -14821.236} C_VEL
LIN {X 0,Y 338.581,Z 368.027,A -85,B 0,C 180,E1 -14822.493,E2 -14822.493} C_VEL
LIN {X 0,Y 339.467,Z 374.48,A -85,B 0,C 180,E1 -14823.118,E2 -14823.118} C_VEL
LIN {X 0,Y 337.419,Z 388.21,A -85,B 0,C 180,E1 -14824.393,E2 -14824.393} C_VEL
LIN {X 0,Y 335.262,Z 401.285,A -85,B 0,C 180,E1 -14825.872,E2 -14825.872} C_VEL
LIN {X 0,Y 333.002,Z 414.421,A -85,B 0,C 180,E1 -14827.673,E2 -14827.673} C_VEL
LIN {X 0,Y 331.111,Z 425.448,A -85,B 0,C 180,E1 -14829.499,E2 -14829.499} C_VEL
LIN {X 0,Y 329.221,Z 436.282,A -85,B 0,C 180,E1 -14831.647,E2 -14831.647} C_VEL
LIN {X 0,Y 327.739,Z 445.324,A -85,B 0,C 180,E1 -14833.813,E2 -14833.813} C_VEL
LIN {X 0,Y 326.522,Z 453.847,A -85,B 0,C 180,E1 -14836.304,E2 -14836.304} C_VEL
LIN {X 0,Y 325.673,Z 460.672,A -85,B 0,C 180,E1 -14838.801,E2 -14838.801} C_VEL
LIN {X 0,Y 325.247,Z 466.008,A -85,B 0,C 180,E1 -14841.3,E2 -14841.3} C_VEL
LIN {X 0,Y 325.066,Z 470.227,A -85,B 0,C 180,E1 -14844.003,E2 -14844.003} C_VEL
LIN {X 0,Y 324.948,Z 472.563,A -85,B 0,C 180,E1 -14846.28,E2 -14846.28} C_VEL
LIN {X 0,Y 325.049,Z 473.941,A -85,B 0,C 180,E1 -14848.761,E2 -14848.761} C_VEL
LIN {X 0,Y 325.019,Z 474.086,A -85,B 0,C 180,E1 -14851.239,E2 -14851.239} C_VEL
LIN {X 0,Y 324.953,Z 473.018,A -85,B 0,C 180,E1 -14853.72,E2 -14853.72} C_VEL
LIN {X 0,Y 325.042,Z 470.741,A -85,B 0,C 180,E1 -14856.206,E2 -14856.206} C_VEL
LIN {X 0,Y 325.236,Z 467.201,A -85,B 0,C 180,E1 -14858.7,E2 -14858.7} C_VEL
LIN {X 0,Y 325.66,Z 462.409,A -85,B 0,C 180,E1 -14861.2,E2 -14861.2} C_VEL
LIN {X 0,Y 326.57,Z 456.307,A -85,B 0,C 180,E1 -14863.694,E2 -14863.694} C_VEL
LIN {X 0,Y 327.878,Z 448.789,A -85,B 0,C 180,E1 -14866.18,E2 -14866.18} C_VEL
LIN {X 0,Y 329.717,Z 439.732,A -85,B 0,C 180,E1 -14868.647,E2 -14868.647} C_VEL
LIN {X 0,Y 332.074,Z 428.95,A -85,B 0,C 180,E1 -14871.087,E2 -14871.087} C_VEL
LIN {X 0,Y 334.745,Z 417.857,A -85,B 0,C 180,E1 -14873.182,E2 -14873.182} C_VEL
LIN {X 0,Y 337.938,Z 404.955,A -85,B 0,C 180,E1 -14875.235,E2 -14875.235} C_VEL
LIN {X 0,Y 341.428,Z 390.97,A -85,B 0,C 180,E1 -14877.092,E2 -14877.092} C_VEL
LIN {X 0,Y 344.318,Z 379.365,A -85,B 0,C 180,E1 -14878.383,E2 -14878.383} C_VEL
LIN {X 0,Y 344.794,Z 367.222,A -85,B 0,C 180,E1 -14879.935,E2 -14879.935} C_VEL
LIN {X 0,Y 344.775,Z 357.945,A -85,B 0,C 180,E1 -14881.114,E2 -14881.114} C_VEL
LIN {X 0,Y 343.554,Z 346.681,A -85,B 0,C 180,E1 -14882.762,E2 -14882.762} C_VEL
LIN {X 0,Y 342.226,Z 339.454,A -85,B 0,C 180,E1 -14883.98,E2 -14883.98} C_VEL
LIN {X 0,Y 340.135,Z 330.691,A -85,B 0,C 180,E1 -14885.742,E2 -14885.742} C_VEL
LIN {X 0,Y 338.791,Z 325.481,A -85,B 0,C 180,E1 -14886.984,E2 -14886.984} C_VEL
LIN {X 0,Y 337.505,Z 321.136,A -85,B 0,C 180,E1 -14888.282,E2 -14888.282} C_VEL
LIN {X 0,Y 337.313,Z 319.574,A -85,B 0,C 180,E1 -14888.687,E2 -14888.687} C_VEL
LIN {X 0,Y 335.657,Z 314.412,A -85,B 0,C 180,E1 -14891.082,E2 -14891.082} C_VEL
LIN {X 0,Y 335.486,Z 311.32,A -85,B 0,C 180,E1 -14892.845,E2 -14892.845} C_VEL
LIN {X 0,Y 335.515,Z 310.568,A -85,B 0,C 180,E1 -14893.729,E2 -14893.729} C_VEL
LIN {X 0,Y 335.864,Z 310.279,A -85,B 0,C 180,E1 -14895.354,E2 -14895.354} C_VEL
LIN {X 0,Y 336.768,Z 310.891,A -85,B 0,C 180,E1 -14896.921,E2 -14896.921} C_VEL
LIN {X 0,Y 338.294,Z 311.744,A -85,B 0,C 180,E1 -14898.409,E2 -14898.409} C_VEL
LIN {X 0,Y 340.363,Z 314.781,A -85,B 0,C 180,E1 -14900.201,E2 -14900.201} C_VEL
LIN {X 0,Y 343.227,Z 319.256,A -85,B 0,C 180,E1 -14902.1,E2 -14902.1} C_VEL
LIN {X 0,Y 346.401,Z 325.399,A -85,B 0,C 180,E1 -14903.959,E2 -14903.959} C_VEL
LIN {X 0,Y 348.75,Z 331.22,A -85,B 0,C 180,E1 -14905.348,E2 -14905.348} C_VEL
LIN {X 0,Y 350.608,Z 337.124,A -85,B 0,C 180,E1 -14906.553,E2 -14906.553} C_VEL
LIN {X 0,Y 350.769,Z 337.908,A -85,B 0,C 180,E1 -14906.688,E2 -14906.688} C_VEL
LIN {X 0,Y 347.194,Z 353.243,A -85,B 0,C 180,E1 -14908.245,E2 -14908.245} C_VEL
LIN {X 0,Y 343.97,Z 366.002,A -85,B 0,C 180,E1 -14909.792,E2 -14909.792} C_VEL
LIN {X 0,Y 341.14,Z 377.064,A -85,B 0,C 180,E1 -14911.381,E2 -14911.381} C_VEL
LIN {X 0,Y 337.979,Z 388.926,A -85,B 0,C 180,E1 -14913.4,E2 -14913.4} C_VEL
LIN {X 0,Y 335.15,Z 399.335,A -85,B 0,C 180,E1 -14915.534,E2 -14915.534} C_VEL
LIN {X 0,Y 332.486,Z 409.061,A -85,B 0,C 180,E1 -14917.964,E2 -14917.964} C_VEL
LIN {X 0,Y 330.577,Z 416.077,A -85,B 0,C 180,E1 -14920.114,E2 -14920.114} C_VEL
LIN {X 0,Y 328.859,Z 422.601,A -85,B 0,C 180,E1 -14922.591,E2 -14922.591} C_VEL
LIN {X 0,Y 327.485,Z 427.658,A -85,B 0,C 180,E1 -14925.077,E2 -14925.077} C_VEL
LIN {X 0,Y 326.464,Z 431.354,A -85,B 0,C 180,E1 -14927.569,E2 -14927.569} C_VEL
LIN {X 0,Y 325.824,Z 433.752,A -85,B 0,C 180,E1 -14930.064,E2 -14930.064} C_VEL
LIN {X 0,Y 325.443,Z 434.909,A -85,B 0,C 180,E1 -14932.555,E2 -14932.555} C_VEL
LIN {X 0,Y 325.274,Z 434.846,A -85,B 0,C 180,E1 -14935.042,E2 -14935.042} C_VEL
LIN {X 0,Y 325.226,Z 433.547,A -85,B 0,C 180,E1 -14937.523,E2 -14937.523} C_VEL
LIN {X 0,Y 325.242,Z 431.016,A -85,B 0,C 180,E1 -14940,E2 -14940} C_VEL
LIN {X 0,Y 325.424,Z 427.189,A -85,B 0,C 180,E1 -14942.476,E2 -14942.476} C_VEL
LIN {X 0,Y 325.941,Z 421.982,A -85,B 0,C 180,E1 -14944.948,E2 -14944.948} C_VEL
LIN {X 0,Y 326.479,Z 415.3,A -85,B 0,C 180,E1 -14947.421,E2 -14947.421} C_VEL
LIN {X 0,Y 327.362,Z 406.95,A -85,B 0,C 180,E1 -14949.89,E2 -14949.89} C_VEL
LIN {X 0,Y 328.517,Z 398.096,A -85,B 0,C 180,E1 -14952.04,E2 -14952.04} C_VEL
LIN {X 0,Y 329.847,Z 387.512,A -85,B 0,C 180,E1 -14954.184,E2 -14954.184} C_VEL
LIN {X 0,Y 331.269,Z 376.779,A -85,B 0,C 180,E1 -14956.01,E2 -14956.01} C_VEL
LIN {X 0,Y 332.91,Z 364.205,A -85,B 0,C 180,E1 -14957.806,E2 -14957.806} C_VEL
LIN {X 0,Y 334.553,Z 350.091,A -85,B 0,C 180,E1 -14959.481,E2 -14959.481} C_VEL
LIN {X 0,Y 336.227,Z 336.344,A -85,B 0,C 180,E1 -14960.815,E2 -14960.815} C_VEL
LIN {X 0,Y 337.42,Z 322.431,A -85,B 0,C 180,E1 -14961.939,E2 -14961.939} C_VEL
LIN {X 0,Y 333.321,Z 306.6,A -85,B 0,C 180,E1 -14963.292,E2 -14963.292} C_VEL
LIN {X 0,Y 328.464,Z 289.908,A -85,B 0,C 180,E1 -14964.491,E2 -14964.491} C_VEL
LIN {X 0,Y 325.681,Z 280.745,A -85,B 0,C 180,E1 -14965.086,E2 -14965.086} C_VEL
LIN {X 0,Y 325.751,Z 279.535,A -85,B 0,C 180,E1 -14966.941,E2 -14966.941} C_VEL
LIN {X 0,Y 326.176,Z 279.477,A -85,B 0,C 180,E1 -14970.473,E2 -14970.473} C_VEL
LIN {X 0,Y 326.472,Z 279.44,A -85,B 0,C 180,E1 -14974.036,E2 -14974.036} C_VEL
LIN {X 0,Y 326.624,Z 279.426,A -85,B 0,C 180,E1 -14977.237,E2 -14977.237} C_VEL
LIN {X 0,Y 326.594,Z 279.425,A -85,B 0,C 180,E1 -14980.209,E2 -14980.209} C_VEL
LIN {X 0,Y 326.565,Z 279.43,A -85,B 0,C 180,E1 -14983.526,E2 -14983.526} C_VEL
LIN {X 0,Y 326.579,Z 279.431,A -85,B 0,C 180,E1 -14987.028,E2 -14987.028} C_VEL
LIN {X 0,Y 326.614,Z 279.428,A -85,B 0,C 180,E1 -14990.773,E2 -14990.773} C_VEL
LIN {X 0,Y 326.616,Z 279.426,A -85,B 0,C 180,E1 -14994.48,E2 -14994.48} C_VEL
LIN {X 0,Y 326.611,Z 279.423,A -85,B 0,C 180,E1 -14997.456,E2 -14997.456} C_VEL
LIN {X 0,Y 326.651,Z 279.421,A -85,B 0,C 180,E1 -15000.34,E2 -15000.34} C_VEL
LIN {X 0,Y 326.693,Z 279.418,A -85,B 0,C 180,E1 -15004.516,E2 -15004.516} C_VEL
LIN {X 0,Y 326.619,Z 279.427,A -85,B 0,C 180,E1 -15008.543,E2 -15008.543} C_VEL
LIN {X 0,Y 326.748,Z 279.406,A -85,B 0,C 180,E1 -15011.178,E2 -15011.178} C_VEL
LIN {X 0,Y 326.766,Z 279.404,A -85,B 0,C 180,E1 -15015.433,E2 -15015.433} C_VEL
LIN {X 0,Y 326.773,Z 279.404,A -85,B 0,C 180,E1 -15018.839,E2 -15018.839} C_VEL
LIN {X 0,Y 326.916,Z 279.387,A -85,B 0,C 180,E1 -15022.589,E2 -15022.589} C_VEL
LIN {X 0,Y 326.761,Z 279.404,A -85,B 0,C 180,E1 -15025.065,E2 -15025.065} C_VEL
LIN {X 0,Y 327.038,Z 279.371,A -85,B 0,C 180,E1 -15027.537,E2 -15027.537} C_VEL
LIN {X 0,Y 327.162,Z 279.36,A -85,B 0,C 180,E1 -15030,E2 -15030} C_VEL
LIN {X 0,Y 327.045,Z 279.37,A -85,B 0,C 180,E1 -15032.463,E2 -15032.463} C_VEL
LIN {X 0,Y 326.954,Z 279.383,A -85,B 0,C 180,E1 -15036.17,E2 -15036.17} C_VEL
LIN {X 0,Y 326.786,Z 279.405,A -85,B 0,C 180,E1 -15039.907,E2 -15039.907} C_VEL
LIN {X 0,Y 326.762,Z 279.41,A -85,B 0,C 180,E1 -15043.685,E2 -15043.685} C_VEL
LIN {X 0,Y 326.703,Z 279.417,A -85,B 0,C 180,E1 -15047.528,E2 -15047.528} C_VEL
LIN {X 0,Y 326.669,Z 279.417,A -85,B 0,C 180,E1 -15050.135,E2 -15050.135} C_VEL
LIN {X 0,Y 326.656,Z 279.418,A -85,B 0,C 180,E1 -15054.129,E2 -15054.129} C_VEL
LIN {X 0,Y 326.686,Z 279.415,A -85,B 0,C 180,E1 -15056.858,E2 -15056.858} C_VEL
LIN {X 0,Y 326.637,Z 279.42,A -85,B 0,C 180,E1 -15060.61,E2 -15060.61} C_VEL
LIN {X 0,Y 326.61,Z 279.423,A -85,B 0,C 180,E1 -15064.019,E2 -15064.019} C_VEL
LIN {X 0,Y 326.626,Z 279.426,A -85,B 0,C 180,E1 -15067.237,E2 -15067.237} C_VEL
LIN {X 0,Y 326.547,Z 279.436,A -85,B 0,C 180,E1 -15071.125,E2 -15071.125} C_VEL
LIN {X 0,Y 326.563,Z 279.43,A -85,B 0,C 180,E1 -15073.526,E2 -15073.526} C_VEL
LIN {X 0,Y 326.579,Z 279.432,A -85,B 0,C 180,E1 -15077.028,E2 -15077.028} C_VEL
LIN {X 0,Y 326.615,Z 279.427,A -85,B 0,C 180,E1 -15080.773,E2 -15080.773} C_VEL
LIN {X 0,Y 326.616,Z 279.425,A -85,B 0,C 180,E1 -15084.48,E2 -15084.48} C_VEL
LIN {X 0,Y 326.611,Z 279.423,A -85,B 0,C 180,E1 -15087.456,E2 -15087.456} C_VEL
LIN {X 0,Y 326.651,Z 279.421,A -85,B 0,C 180,E1 -15090.34,E2 -15090.34} C_VEL
LIN {X 0,Y 326.693,Z 279.418,A -85,B 0,C 180,E1 -15094.516,E2 -15094.516} C_VEL
LIN {X 0,Y 326.623,Z 279.427,A -85,B 0,C 180,E1 -15098.543,E2 -15098.543} C_VEL
LIN {X 0,Y 326.631,Z 279.42,A -85,B 0,C 180,E1 -15099.46,E2 -15099.46} C_VEL
LIN {X 0,Y 326.011,Z 279.503,A -85,B 0,C 180,E1 -15100.489,E2 -15100.489} C_VEL
LIN {X 0,Y 323.184,Z 279.855,A -85,B 0,C 180,E1 -15102.165,E2 -15102.165} C_VEL
LIN {X 0,Y 320.782,Z 280.154,A -85,B 0,C 180,E1 -15103.522,E2 -15103.522} C_VEL
LIN {X 0,Y 319.778,Z 280.277,A -85,B 0,C 180,E1 -15104.573,E2 -15104.573} C_VEL
LIN {X 0,Y 319.712,Z 280.283,A -85,B 0,C 180,E1 -15104.929,E2 -15104.929} C_VEL
LIN {X 0,Y 319.719,Z 280.284,A -85,B 0,C 180,E1 -15108.589,E2 -15108.589} C_VEL
LIN {X 0,Y 319.857,Z 280.267,A -85,B 0,C 180,E1 -15112.424,E2 -15112.424} C_VEL
LIN {X 0,Y 319.732,Z 280.28,A -85,B 0,C 180,E1 -15114.956,E2 -15114.956} C_VEL
LIN {X 0,Y 319.989,Z 280.249,A -85,B 0,C 180,E1 -15117.482,E2 -15117.482} C_VEL
LIN {X 0,Y 320.099,Z 280.24,A -85,B 0,C 180,E1 -15120,E2 -15120} C_VEL
LIN {X 0,Y 319.993,Z 280.248,A -85,B 0,C 180,E1 -15122.517,E2 -15122.517} C_VEL
LIN {X 0,Y 319.906,Z 280.26,A -85,B 0,C 180,E1 -15126.306,E2 -15126.306} C_VEL
LIN {X 0,Y 319.739,Z 280.281,A -85,B 0,C 180,E1 -15130.127,E2 -15130.127} C_VEL
LIN {X 0,Y 319.735,Z 280.282,A -85,B 0,C 180,E1 -15133.992,E2 -15133.992} C_VEL
LIN {X 0,Y 319.661,Z 280.291,A -85,B 0,C 180,E1 -15137.926,E2 -15137.926} C_VEL
LIN {X 0,Y 319.619,Z 280.294,A -85,B 0,C 180,E1 -15140.598,E2 -15140.598} C_VEL
LIN {X 0,Y 319.566,Z 280.304,A -85,B 0,C 180,E1 -15143.319,E2 -15143.319} C_VEL
LIN {X 0,Y 319.572,Z 280.304,A -85,B 0,C 180,E1 -15146.093,E2 -15146.093} C_VEL
LIN {X 0,Y 319.545,Z 280.307,A -85,B 0,C 180,E1 -15148.938,E2 -15148.938} C_VEL
LIN {X 0,Y 319.583,Z 280.435,A -85,B 0,C 180,E1 -15150.945,E2 -15150.945} C_VEL
LIN {X 0,Y 320.344,Z 284.871,A -85,B 0,C 180,E1 -15154.779,E2 -15154.779} C_VEL
LIN {X 0,Y 321.036,Z 288.813,A -85,B 0,C 180,E1 -15157.991,E2 -15157.991} C_VEL
LIN {X 0,Y 322.068,Z 294.153,A -85,B 0,C 180,E1 -15162.103,E2 -15162.103} C_VEL
LIN {X 0,Y 322.95,Z 299.41,A -85,B 0,C 180,E1 -15165.901,E2 -15165.901} C_VEL
LIN {X 0,Y 323.038,Z 303.203,A -85,B 0,C 180,E1 -15168.471,E2 -15168.471} C_VEL
LIN {X 0,Y 322.37,Z 308.262,A -85,B 0,C 180,E1 -15171.705,E2 -15171.705} C_VEL
LIN {X 0,Y 321.473,Z 314.183,A -85,B 0,C 180,E1 -15175.36,E2 -15175.36} C_VEL
LIN {X 0,Y 320.858,Z 318.97,A -85,B 0,C 180,E1 -15178.239,E2 -15178.239} C_VEL
LIN {X 0,Y 325.367,Z 337.644,A -85,B 0,C 180,E1 -15179.465,E2 -15179.465} C_VEL
LIN {X 0,Y 329.084,Z 354.423,A -85,B 0,C 180,E1 -15180.801,E2 -15180.801} C_VEL
LIN {X 0,Y 331.741,Z 368.661,A -85,B 0,C 180,E1 -15182.113,E2 -15182.113} C_VEL
LIN {X 0,Y 332.655,Z 374.887,A -85,B 0,C 180,E1 -15182.741,E2 -15182.741} C_VEL
LIN {X 0,Y 330.948,Z 386.569,A -85,B 0,C 180,E1 -15183.855,E2 -15183.855} C_VEL
LIN {X 0,Y 328.627,Z 399.806,A -85,B 0,C 180,E1 -15185.353,E2 -15185.353} C_VEL
LIN {X 0,Y 326.508,Z 412.07,A -85,B 0,C 180,E1 -15187.037,E2 -15187.037} C_VEL
LIN {X 0,Y 324.461,Z 423.322,A -85,B 0,C 180,E1 -15188.882,E2 -15188.882} C_VEL
LIN {X 0,Y 322.684,Z 433.757,A -85,B 0,C 180,E1 -15190.931,E2 -15190.931} C_VEL
LIN {X 0,Y 321.032,Z 443.135,A -85,B 0,C 180,E1 -15193.138,E2 -15193.138} C_VEL
LIN {X 0,Y 319.748,Z 451.191,A -85,B 0,C 180,E1 -15195.428,E2 -15195.428} C_VEL
LIN {X 0,Y 318.891,Z 458.307,A -85,B 0,C 180,E1 -15197.914,E2 -15197.914} C_VEL
LIN {X 0,Y 318.241,Z 464.068,A -85,B 0,C 180,E1 -15200.466,E2 -15200.466} C_VEL
LIN {X 0,Y 318.04,Z 467.483,A -85,B 0,C 180,E1 -15202.381,E2 -15202.381} C_VEL
LIN {X 0,Y 317.994,Z 469.799,A -85,B 0,C 180,E1 -15204.012,E2 -15204.012} C_VEL
LIN {X 0,Y 317.879,Z 472.005,A -85,B 0,C 180,E1 -15206.197,E2 -15206.197} C_VEL
LIN {X 0,Y 317.959,Z 473.447,A -85,B 0,C 180,E1 -15208.733,E2 -15208.733} C_VEL
LIN {X 0,Y 317.992,Z 473.707,A -85,B 0,C 180,E1 -15210,E2 -15210} C_VEL
LIN {X 0,Y 317.852,Z 473.303,A -85,B 0,C 180,E1 -15212.535,E2 -15212.535} C_VEL
LIN {X 0,Y 317.87,Z 471.686,A -85,B 0,C 180,E1 -15215.074,E2 -15215.074} C_VEL
LIN {X 0,Y 317.996,Z 468.823,A -85,B 0,C 180,E1 -15217.62,E2 -15217.62} C_VEL
LIN {X 0,Y 318.353,Z 464.748,A -85,B 0,C 180,E1 -15220.172,E2 -15220.172} C_VEL
LIN {X 0,Y 319.12,Z 459.419,A -85,B 0,C 180,E1 -15222.723,E2 -15222.723} C_VEL
LIN {X 0,Y 320.254,Z 452.753,A -85,B 0,C 180,E1 -15225.268,E2 -15225.268} C_VEL
LIN {X 0,Y 321.924,Z 444.651,A -85,B 0,C 180,E1 -15227.797,E2 -15227.797} C_VEL
LIN {X 0,Y 324.147,Z 434.969,A -85,B 0,C 180,E1 -15230.298,E2 -15230.298} C_VEL
LIN {X 0,Y 326.569,Z 425.305,A -85,B 0,C 180,E1 -15232.403,E2 -15232.403} C_VEL
LIN {X 0,Y 329.661,Z 413.551,A -85,B 0,C 180,E1 -15234.565,E2 -15234.565} C_VEL
LIN {X 0,Y 332.976,Z 401.228,A -85,B 0,C 180,E1 -15236.48,E2 -15236.48} C_VEL
LIN {X 0,Y 336.571,Z 388.105,A -85,B 0,C 180,E1 -15238.193,E2 -15238.193} C_VEL
LIN {X 0,Y 338.617,Z 380.09,A -85,B 0,C 180,E1 -15239.116,E2 -15239.116} C_VEL
LIN {X 0,Y 339.502,Z 362.626,A -85,B 0,C 180,E1 -15241.479,E2 -15241.479} C_VEL
LIN {X 0,Y 338.902,Z 352.352,A -85,B 0,C 180,E1 -15243.042,E2 -15243.042} C_VEL
LIN {X 0,Y 337.822,Z 344.195,A -85,B 0,C 180,E1 -15244.47,E2 -15244.47} C_VEL
LIN {X 0,Y 336.361,Z 336.555,A -85,B 0,C 180,E1 -15246.068,E2 -15246.068} C_VEL
LIN {X 0,Y 335.184,Z 330.973,A -85,B 0,C 180,E1 -15247.45,E2 -15247.45} C_VEL
LIN {X 0,Y 334.165,Z 326.218,A -85,B 0,C 180,E1 -15248.907,E2 -15248.907} C_VEL
LIN {X 0,Y 334.098,Z 325.38,A -85,B 0,C 180,E1 -15249.13,E2 -15249.13} C_VEL
LIN {X 0,Y 332.866,Z 320.304,A -85,B 0,C 180,E1 -15251.594,E2 -15251.594} C_VEL
LIN {X 0,Y 332.848,Z 318.677,A -85,B 0,C 180,E1 -15252.507,E2 -15252.507} C_VEL
LIN {X 0,Y 333.01,Z 317.04,A -85,B 0,C 180,E1 -15254.148,E2 -15254.148} C_VEL
LIN {X 0,Y 333.522,Z 317.063,A -85,B 0,C 180,E1 -15255.943,E2 -15255.943} C_VEL
LIN {X 0,Y 334.928,Z 317.927,A -85,B 0,C 180,E1 -15257.819,E2 -15257.819} C_VEL
LIN {X 0,Y 336.742,Z 320.534,A -85,B 0,C 180,E1 -15259.685,E2 -15259.685} C_VEL
LIN {X 0,Y 338.488,Z 323.369,A -85,B 0,C 180,E1 -15261.07,E2 -15261.07} C_VEL
LIN {X 0,Y 339.877,Z 325.755,A -85,B 0,C 180,E1 -15262.05,E2 -15262.05} C_VEL
LIN {X 0,Y 342.332,Z 331.056,A -85,B 0,C 180,E1 -15263.713,E2 -15263.713} C_VEL
LIN {X 0,Y 344.387,Z 336.863,A -85,B 0,C 180,E1 -15265.152,E2 -15265.152} C_VEL
LIN {X 0,Y 345.398,Z 340.392,A -85,B 0,C 180,E1 -15265.913,E2 -15265.913} C_VEL
LIN {X 0,Y 345.021,Z 342.774,A -85,B 0,C 180,E1 -15266.202,E2 -15266.202} C_VEL
LIN {X 0,Y 341.57,Z 356.265,A -85,B 0,C 180,E1 -15267.659,E2 -15267.659} C_VEL
LIN {X 0,Y 337.919,Z 369.581,A -85,B 0,C 180,E1 -15269.367,E2 -15269.367} C_VEL
LIN {X 0,Y 334.171,Z 382.73,A -85,B 0,C 180,E1 -15271.415,E2 -15271.415} C_VEL
LIN {X 0,Y 330.9,Z 393.862,A -85,B 0,C 180,E1 -15273.512,E2 -15273.512} C_VEL
LIN {X 0,Y 328.092,Z 403.314,A -85,B 0,C 180,E1 -15275.648,E2 -15275.648} C_VEL
LIN {X 0,Y 325.689,Z 411.338,A -85,B 0,C 180,E1 -15277.814,E2 -15277.814} C_VEL
LIN {X 0,Y 323.438,Z 418.873,A -85,B 0,C 180,E1 -15280.318,E2 -15280.318} C_VEL
LIN {X 0,Y 321.686,Z 424.879,A -85,B 0,C 180,E1 -15282.846,E2 -15282.846} C_VEL
LIN {X 0,Y 320.652,Z 428.502,A -85,B 0,C 180,E1 -15284.751,E2 -15284.751} C_VEL
LIN {X 0,Y 319.524,Z 432.097,A -85,B 0,C 180,E1 -15287.294,E2 -15287.294} C_VEL
LIN {X 0,Y 318.827,Z 434.41,A -85,B 0,C 180,E1 -15289.843,E2 -15289.843} C_VEL
LIN {X 0,Y 318.391,Z 435.494,A -85,B 0,C 180,E1 -15292.39,E2 -15292.39} C_VEL
LIN {X 0,Y 318.218,Z 435.345,A -85,B 0,C 180,E1 -15294.932,E2 -15294.932} C_VEL
LIN {X 0,Y 318.132,Z 433.98,A -85,B 0,C 180,E1 -15297.468,E2 -15297.468} C_VEL
LIN {X 0,Y 318.15,Z 431.369,A -85,B 0,C 180,E1 -15300,E2 -15300} C_VEL
LIN {X 0,Y 318.337,Z 427.467,A -85,B 0,C 180,E1 -15302.531,E2 -15302.531} C_VEL
LIN {X 0,Y 318.872,Z 422.198,A -85,B 0,C 180,E1 -15305.058,E2 -15305.058} C_VEL
LIN {X 0,Y 319.439,Z 415.431,A -85,B 0,C 180,E1 -15307.586,E2 -15307.586} C_VEL
LIN {X 0,Y 320.361,Z 406.981,A -85,B 0,C 180,E1 -15310.108,E2 -15310.108} C_VEL
LIN {X 0,Y 321.572,Z 398.023,A -85,B 0,C 180,E1 -15312.304,E2 -15312.304} C_VEL
LIN {X 0,Y 322.944,Z 387.32,A -85,B 0,C 180,E1 -15314.494,E2 -15314.494} C_VEL
LIN {X 0,Y 324.423,Z 376.456,A -85,B 0,C 180,E1 -15316.357,E2 -15316.357} C_VEL
LIN {X 0,Y 326.056,Z 364.164,A -85,B 0,C 180,E1 -15318.135,E2 -15318.135} C_VEL
LIN {X 0,Y 327.667,Z 350.892,A -85,B 0,C 180,E1 -15319.744,E2 -15319.744} C_VEL
LIN {X 0,Y 329.348,Z 337.289,A -85,B 0,C 180,E1 -15321.107,E2 -15321.107} C_VEL
LIN {X 0,Y 330.567,Z 323.663,A -85,B 0,C 180,E1 -15322.247,E2 -15322.247} C_VEL
LIN {X 0,Y 326.586,Z 308.174,A -85,B 0,C 180,E1 -15323.605,E2 -15323.605} C_VEL
LIN {X 0,Y 322.063,Z 292.391,A -85,B 0,C 180,E1 -15324.793,E2 -15324.793} C_VEL
LIN {X 0,Y 318.625,Z 281.171,A -85,B 0,C 180,E1 -15325.551,E2 -15325.551} C_VEL
LIN {X 0,Y 318.638,Z 280.629,A -85,B 0,C 180,E1 -15326.176,E2 -15326.176} C_VEL
LIN {X 0,Y 318.955,Z 280.381,A -85,B 0,C 180,E1 -15328.997,E2 -15328.997} C_VEL
LIN {X 0,Y 319.239,Z 280.342,A -85,B 0,C 180,E1 -15331.895,E2 -15331.895} C_VEL
LIN {X 0,Y 319.533,Z 280.307,A -85,B 0,C 180,E1 -15335.531,E2 -15335.531} C_VEL
LIN {X 0,Y 319.542,Z 280.304,A -85,B 0,C 180,E1 -15338.013,E2 -15338.013} C_VEL
LIN {X 0,Y 319.528,Z 280.306,A -85,B 0,C 180,E1 -15341.597,E2 -15341.597} C_VEL
LIN {X 0,Y 319.491,Z 280.313,A -85,B 0,C 180,E1 -15345.257,E2 -15345.257} C_VEL
LIN {X 0,Y 319.532,Z 280.309,A -85,B 0,C 180,E1 -15348.712,E2 -15348.712} C_VEL
LIN {X 0,Y 319.557,Z 280.303,A -85,B 0,C 180,E1 -15352.35,E2 -15352.35} C_VEL
LIN {X 0,Y 319.563,Z 280.303,A -85,B 0,C 180,E1 -15355.124,E2 -15355.124} C_VEL
LIN {X 0,Y 319.569,Z 280.302,A -85,B 0,C 180,E1 -15359.059,E2 -15359.059} C_VEL
LIN {X 0,Y 319.609,Z 280.3,A -85,B 0,C 180,E1 -15362.498,E2 -15362.498} C_VEL
LIN {X 0,Y 319.605,Z 280.296,A -85,B 0,C 180,E1 -15365.304,E2 -15365.304} C_VEL
LIN {X 0,Y 319.602,Z 280.296,A -85,B 0,C 180,E1 -15369.4,E2 -15369.4} C_VEL
LIN {X 0,Y 319.662,Z 280.292,A -85,B 0,C 180,E1 -15372.073,E2 -15372.073} C_VEL
LIN {X 0,Y 319.735,Z 280.282,A -85,B 0,C 180,E1 -15376.008,E2 -15376.008} C_VEL
LIN {X 0,Y 319.755,Z 280.28,A -85,B 0,C 180,E1 -15379.873,E2 -15379.873} C_VEL
LIN {X 0,Y 319.904,Z 280.26,A -85,B 0,C 180,E1 -15383.694,E2 -15383.694} C_VEL
LIN {X 0,Y 319.981,Z 280.25,A -85,B 0,C 180,E1 -15387.482,E2 -15387.482} C_VEL
LIN {X 0,Y 320.115,Z 280.237,A -85,B 0,C 180,E1 -15390,E2 -15390} C_VEL
LIN {X 0,Y 319.989,Z 280.249,A -85,B 0,C 180,E1 -15392.518,E2 -15392.518} C_VEL
LIN {X 0,Y 319.91,Z 280.259,A -85,B 0,C 180,E1 -15396.306,E2 -15396.306} C_VEL
LIN {X 0,Y 319.739,Z 280.281,A -85,B 0,C 180,E1 -15400.128,E2 -15400.128} C_VEL
LIN {X 0,Y 319.735,Z 280.282,A -85,B 0,C 180,E1 -15403.992,E2 -15403.992} C_VEL
LIN {X 0,Y 319.662,Z 280.291,A -85,B 0,C 180,E1 -15407.927,E2 -15407.927} C_VEL
LIN {X 0,Y 319.619,Z 280.294,A -85,B 0,C 180,E1 -15410.599,E2 -15410.599} C_VEL
LIN {X 0,Y 319.574,Z 280.304,A -85,B 0,C 180,E1 -15413.319,E2 -15413.319} C_VEL
LIN {X 0,Y 319.621,Z 280.294,A -85,B 0,C 180,E1 -15416.089,E2 -15416.089} C_VEL
LIN {X 0,Y 319.583,Z 280.3,A -85,B 0,C 180,E1 -15418.934,E2 -15418.934} C_VEL
LIN {X 0,Y 319.534,Z 280.305,A -85,B 0,C 180,E1 -15421.862,E2 -15421.862} C_VEL
LIN {X 0,Y 319.583,Z 280.301,A -85,B 0,C 180,E1 -15425.543,E2 -15425.543} C_VEL
LIN {X 0,Y 319.53,Z 280.306,A -85,B 0,C 180,E1 -15429.662,E2 -15429.662} C_VEL
LIN {X 0,Y 319.522,Z 280.308,A -85,B 0,C 180,E1 -15433.46,E2 -15433.46} C_VEL
LIN {X 0,Y 319.557,Z 280.307,A -85,B 0,C 180,E1 -15437.016,E2 -15437.016} C_VEL
LIN {X 0,Y 319.55,Z 280.304,A -85,B 0,C 180,E1 -15440.371,E2 -15440.371} C_VEL
LIN {X 0,Y 319.584,Z 280.301,A -85,B 0,C 180,E1 -15444.457,E2 -15444.457} C_VEL
LIN {X 0,Y 319.534,Z 280.305,A -85,B 0,C 180,E1 -15448.138,E2 -15448.138} C_VEL
LIN {X 0,Y 319.614,Z 280.294,A -85,B 0,C 180,E1 -15451.59,E2 -15451.59} C_VEL
LIN {X 0,Y 319.607,Z 280.296,A -85,B 0,C 180,E1 -15455.304,E2 -15455.304} C_VEL
LIN {X 0,Y 319.605,Z 280.295,A -85,B 0,C 180,E1 -15459.459,E2 -15459.459} C_VEL
LIN {X 0,Y 319.663,Z 280.291,A -85,B 0,C 180,E1 -15462.073,E2 -15462.073} C_VEL
LIN {X 0,Y 319.712,Z 280.283,A -85,B 0,C 180,E1 -15464.929,E2 -15464.929} C_VEL
LIN {X 0,Y 319.077,Z 280.366,A -85,B 0,C 180,E1 -15465.981,E2 -15465.981} C_VEL
LIN {X 0,Y 316.207,Z 280.72,A -85,B 0,C 180,E1 -15467.692,E2 -15467.692} C_VEL
LIN {X 0,Y 313.778,Z 281.022,A -85,B 0,C 180,E1 -15469.079,E2 -15469.079} C_VEL
LIN {X 0,Y 312.774,Z 281.151,A -85,B 0,C 180,E1 -15470.154,E2 -15470.154} C_VEL
LIN {X 0,Y 312.715,Z 281.152,A -85,B 0,C 180,E1 -15470.517,E2 -15470.517} C_VEL
LIN {X 0,Y 312.846,Z 281.138,A -85,B 0,C 180,E1 -15473.55,E2 -15473.55} C_VEL
LIN {X 0,Y 312.935,Z 281.127,A -85,B 0,C 180,E1 -15477.425,E2 -15477.425} C_VEL
LIN {X 0,Y 313.055,Z 281.117,A -85,B 0,C 180,E1 -15480,E2 -15480} C_VEL
LIN {X 0,Y 312.939,Z 281.127,A -85,B 0,C 180,E1 -15482.574,E2 -15482.574} C_VEL
LIN {X 0,Y 312.847,Z 281.138,A -85,B 0,C 180,E1 -15486.449,E2 -15486.449} C_VEL
LIN {X 0,Y 312.754,Z 281.149,A -85,B 0,C 180,E1 -15489.05,E2 -15489.05} C_VEL
LIN {X 0,Y 312.637,Z 281.164,A -85,B 0,C 180,E1 -15492.991,E2 -15492.991} C_VEL
LIN {X 0,Y 312.641,Z 281.169,A -85,B 0,C 180,E1 -15495.649,E2 -15495.649} C_VEL
LIN {X 0,Y 312.633,Z 281.166,A -85,B 0,C 180,E1 -15499.236,E2 -15499.236} C_VEL
LIN {X 0,Y 312.546,Z 281.176,A -85,B 0,C 180,E1 -15502.788,E2 -15502.788} C_VEL
LIN {X 0,Y 312.532,Z 281.181,A -85,B 0,C 180,E1 -15505.908,E2 -15505.908} C_VEL
LIN {X 0,Y 312.5,Z 281.184,A -85,B 0,C 180,E1 -15509.654,E2 -15509.654} C_VEL
LIN {X 0,Y 312.532,Z 281.207,A -85,B 0,C 180,E1 -15510.395,E2 -15510.395} C_VEL
LIN {X 0,Y 313.228,Z 285.413,A -85,B 0,C 180,E1 -15514.12,E2 -15514.12} C_VEL
LIN {X 0,Y 313.846,Z 289.096,A -85,B 0,C 180,E1 -15517.201,E2 -15517.201} C_VEL
LIN {X 0,Y 314.661,Z 293.34,A -85,B 0,C 180,E1 -15520.589,E2 -15520.589} C_VEL
LIN {X 0,Y 315.428,Z 297.421,A -85,B 0,C 180,E1 -15523.686,E2 -15523.686} C_VEL
LIN {X 0,Y 316.016,Z 301.201,A -85,B 0,C 180,E1 -15526.415,E2 -15526.415} C_VEL
LIN {X 0,Y 316.043,Z 303.732,A -85,B 0,C 180,E1 -15528.154,E2 -15528.154} C_VEL
LIN {X 0,Y 315.375,Z 308.669,A -85,B 0,C 180,E1 -15531.393,E2 -15531.393} C_VEL
LIN {X 0,Y 314.441,Z 314.726,A -85,B 0,C 180,E1 -15535.218,E2 -15535.218} C_VEL
LIN {X 0,Y 313.948,Z 318.648,A -85,B 0,C 180,E1 -15537.646,E2 -15537.646} C_VEL
LIN {X 0,Y 318.62,Z 338.355,A -85,B 0,C 180,E1 -15538.99,E2 -15538.99} C_VEL
LIN {X 0,Y 322.221,Z 355.032,A -85,B 0,C 180,E1 -15540.367,E2 -15540.367} C_VEL
LIN {X 0,Y 324.829,Z 369.039,A -85,B 0,C 180,E1 -15541.707,E2 -15541.707} C_VEL
LIN {X 0,Y 325.785,Z 376.675,A -85,B 0,C 180,E1 -15542.5,E2 -15542.5} C_VEL
LIN {X 0,Y 323.746,Z 389.172,A -85,B 0,C 180,E1 -15543.749,E2 -15543.749} C_VEL
LIN {X 0,Y 321.509,Z 401.918,A -85,B 0,C 180,E1 -15545.288,E2 -15545.288} C_VEL
LIN {X 0,Y 319.293,Z 413.759,A -85,B 0,C 180,E1 -15547.002,E2 -15547.002} C_VEL
LIN {X 0,Y 317.234,Z 425.092,A -85,B 0,C 180,E1 -15548.968,E2 -15548.968} C_VEL
LIN {X 0,Y 315.315,Z 435.543,A -85,B 0,C 180,E1 -15551.144,E2 -15551.144} C_VEL
LIN {X 0,Y 313.742,Z 444.562,A -85,B 0,C 180,E1 -15553.405,E2 -15553.405} C_VEL
LIN {X 0,Y 312.543,Z 452.073,A -85,B 0,C 180,E1 -15555.679,E2 -15555.679} C_VEL
LIN {X 0,Y 311.643,Z 459.092,A -85,B 0,C 180,E1 -15558.29,E2 -15558.29} C_VEL
LIN {X 0,Y 311.107,Z 464.578,A -85,B 0,C 180,E1 -15560.901,E2 -15560.901} C_VEL
LIN {X 0,Y 310.89,Z 468.666,A -85,B 0,C 180,E1 -15563.51,E2 -15563.51} C_VEL
LIN {X 0,Y 310.812,Z 471.431,A -85,B 0,C 180,E1 -15566.11,E2 -15566.11} C_VEL
LIN {X 0,Y 310.869,Z 472.943,A -85,B 0,C 180,E1 -15568.705,E2 -15568.705} C_VEL
LIN {X 0,Y 310.907,Z 473.24,A -85,B 0,C 180,E1 -15570,E2 -15570} C_VEL
LIN {X 0,Y 310.77,Z 472.906,A -85,B 0,C 180,E1 -15572.592,E2 -15572.592} C_VEL
LIN {X 0,Y 310.793,Z 471.323,A -85,B 0,C 180,E1 -15575.19,E2 -15575.19} C_VEL
LIN {X 0,Y 310.916,Z 468.544,A -85,B 0,C 180,E1 -15577.795,E2 -15577.795} C_VEL
LIN {X 0,Y 311.309,Z 464.563,A -85,B 0,C 180,E1 -15580.405,E2 -15580.405} C_VEL
LIN {X 0,Y 312.139,Z 459.353,A -85,B 0,C 180,E1 -15583.012,E2 -15583.012} C_VEL
LIN {X 0,Y 313.354,Z 452.829,A -85,B 0,C 180,E1 -15585.613,E2 -15585.613} C_VEL
LIN {X 0,Y 315.145,Z 444.908,A -85,B 0,C 180,E1 -15588.193,E2 -15588.193} C_VEL
LIN {X 0,Y 317.485,Z 435.458,A -85,B 0,C 180,E1 -15590.744,E2 -15590.744} C_VEL
LIN {X 0,Y 320.027,Z 426.144,A -85,B 0,C 180,E1 -15592.862,E2 -15592.862} C_VEL
LIN {X 0,Y 323.296,Z 414.659,A -85,B 0,C 180,E1 -15595.081,E2 -15595.081} C_VEL
LIN {X 0,Y 327.077,Z 401.799,A -85,B 0,C 180,E1 -15597.168,E2 -15597.168} C_VEL
LIN {X 0,Y 331.192,Z 387.913,A -85,B 0,C 180,E1 -15599.04,E2 -15599.04} C_VEL
LIN {X 0,Y 332.864,Z 382.13,A -85,B 0,C 180,E1 -15599.732,E2 -15599.732} C_VEL
LIN {X 0,Y 334.201,Z 364.818,A -85,B 0,C 180,E1 -15602.215,E2 -15602.215} C_VEL
LIN {X 0,Y 333.889,Z 354.726,A -85,B 0,C 180,E1 -15603.867,E2 -15603.867} C_VEL
LIN {X 0,Y 333.099,Z 347.101,A -85,B 0,C 180,E1 -15605.333,E2 -15605.333} C_VEL
LIN {X 0,Y 332.061,Z 340.263,A -85,B 0,C 180,E1 -15606.914,E2 -15606.914} C_VEL
LIN {X 0,Y 331.487,Z 336.354,A -85,B 0,C 180,E1 -15607.941,E2 -15607.941} C_VEL
LIN {X 0,Y 330.753,Z 331.073,A -85,B 0,C 180,E1 -15609.603,E2 -15609.603} C_VEL
LIN {X 0,Y 329.965,Z 326.735,A -85,B 0,C 180,E1 -15611.801,E2 -15611.801} C_VEL
LIN {X 0,Y 330.047,Z 324.832,A -85,B 0,C 180,E1 -15612.954,E2 -15612.954} C_VEL
LIN {X 0,Y 330.323,Z 323.557,A -85,B 0,C 180,E1 -15614.597,E2 -15614.597} C_VEL
LIN {X 0,Y 330.882,Z 323.694,A -85,B 0,C 180,E1 -15616.234,E2 -15616.234} C_VEL
LIN {X 0,Y 332.012,Z 324.444,A -85,B 0,C 180,E1 -15617.806,E2 -15617.806} C_VEL
LIN {X 0,Y 334.238,Z 327.905,A -85,B 0,C 180,E1 -15620.194,E2 -15620.194} C_VEL
LIN {X 0,Y 336.527,Z 332.532,A -85,B 0,C 180,E1 -15622.139,E2 -15622.139} C_VEL
LIN {X 0,Y 338.841,Z 338.585,A -85,B 0,C 180,E1 -15623.99,E2 -15623.99} C_VEL
LIN {X 0,Y 340.323,Z 344.124,A -85,B 0,C 180,E1 -15625.333,E2 -15625.333} C_VEL
LIN {X 0,Y 336.421,Z 358.02,A -85,B 0,C 180,E1 -15626.888,E2 -15626.888} C_VEL
LIN {X 0,Y 332.789,Z 370.153,A -85,B 0,C 180,E1 -15628.488,E2 -15628.488} C_VEL
LIN {X 0,Y 328.788,Z 383.142,A -85,B 0,C 180,E1 -15630.552,E2 -15630.552} C_VEL
LIN {X 0,Y 325.365,Z 393.789,A -85,B 0,C 180,E1 -15632.58,E2 -15632.58} C_VEL
LIN {X 0,Y 322.178,Z 403.595,A -85,B 0,C 180,E1 -15634.826,E2 -15634.826} C_VEL
LIN {X 0,Y 319.571,Z 411.573,A -85,B 0,C 180,E1 -15637.024,E2 -15637.024} C_VEL
LIN {X 0,Y 317.345,Z 418.319,A -85,B 0,C 180,E1 -15639.247,E2 -15639.247} C_VEL
LIN {X 0,Y 315.394,Z 424.526,A -85,B 0,C 180,E1 -15641.823,E2 -15641.823} C_VEL
LIN {X 0,Y 313.791,Z 429.361,A -85,B 0,C 180,E1 -15644.41,E2 -15644.41} C_VEL
LIN {X 0,Y 312.594,Z 432.867,A -85,B 0,C 180,E1 -15647.008,E2 -15647.008} C_VEL
LIN {X 0,Y 311.826,Z 435.085,A -85,B 0,C 180,E1 -15649.613,E2 -15649.613} C_VEL
LIN {X 0,Y 311.336,Z 436.079,A -85,B 0,C 180,E1 -15652.216,E2 -15652.216} C_VEL
LIN {X 0,Y 311.163,Z 435.851,A -85,B 0,C 180,E1 -15654.817,E2 -15654.817} C_VEL
LIN {X 0,Y 311.038,Z 434.402,A -85,B 0,C 180,E1 -15657.41,E2 -15657.41} C_VEL
LIN {X 0,Y 311.058,Z 431.715,A -85,B 0,C 180,E1 -15660,E2 -15660} C_VEL
LIN {X 0,Y 311.25,Z 427.728,A -85,B 0,C 180,E1 -15662.589,E2 -15662.589} C_VEL
LIN {X 0,Y 311.808,Z 422.361,A -85,B 0,C 180,E1 -15665.173,E2 -15665.173} C_VEL
LIN {X 0,Y 312.375,Z 415.508,A -85,B 0,C 180,E1 -15667.758,E2 -15667.758} C_VEL
LIN {X 0,Y 313.362,Z 406.98,A -85,B 0,C 180,E1 -15670.336,E2 -15670.336} C_VEL
LIN {X 0,Y 314.636,Z 397.938,A -85,B 0,C 180,E1 -15672.579,E2 -15672.579} C_VEL
LIN {X 0,Y 316.048,Z 387.118,A -85,B 0,C 180,E1 -15674.817,E2 -15674.817} C_VEL
LIN {X 0,Y 317.598,Z 376.128,A -85,B 0,C 180,E1 -15676.719,E2 -15676.719} C_VEL
LIN {X 0,Y 319.379,Z 362.876,A -85,B 0,C 180,E1 -15678.644,E2 -15678.644} C_VEL
LIN {X 0,Y 321.118,Z 348.874,A -85,B 0,C 180,E1 -15680.331,E2 -15680.331} C_VEL
LIN {X 0,Y 322.894,Z 334.801,A -85,B 0,C 180,E1 -15681.717,E2 -15681.717} C_VEL
LIN {X 0,Y 323.732,Z 325.038,A -85,B 0,C 180,E1 -15682.537,E2 -15682.537} C_VEL
LIN {X 0,Y 319.926,Z 310.051,A -85,B 0,C 180,E1 -15683.906,E2 -15683.906} C_VEL
LIN {X 0,Y 315.312,Z 293.784,A -85,B 0,C 180,E1 -15685.187,E2 -15685.187} C_VEL
LIN {X 0,Y 311.586,Z 281.555,A -85,B 0,C 180,E1 -15686.03,E2 -15686.03} C_VEL
LIN {X 0,Y 311.654,Z 281.291,A -85,B 0,C 180,E1 -15686.809,E2 -15686.809} C_VEL
LIN {X 0,Y 311.984,Z 281.247,A -85,B 0,C 180,E1 -15689.709,E2 -15689.709} C_VEL
LIN {X 0,Y 312.343,Z 281.202,A -85,B 0,C 180,E1 -15693.64,E2 -15693.64} C_VEL
LIN {X 0,Y 312.502,Z 281.181,A -85,B 0,C 180,E1 -15695.941,E2 -15695.941} C_VEL
LIN {X 0,Y 312.5,Z 281.186,A -85,B 0,C 180,E1 -15699.029,E2 -15699.029} C_VEL
LIN {X 0,Y 312.493,Z 281.183,A -85,B 0,C 180,E1 -15702.432,E2 -15702.432} C_VEL
LIN {X 0,Y 312.461,Z 281.186,A -85,B 0,C 180,E1 -15706.035,E2 -15706.035} C_VEL
LIN {X 0,Y 312.507,Z 281.18,A -85,B 0,C 180,E1 -15709.875,E2 -15709.875} C_VEL
LIN {X 0,Y 312.538,Z 281.176,A -85,B 0,C 180,E1 -15714.05,E2 -15714.05} C_VEL
LIN {X 0,Y 312.506,Z 281.181,A -85,B 0,C 180,E1 -15717.334,E2 -15717.334} C_VEL
LIN {X 0,Y 312.547,Z 281.175,A -85,B 0,C 180,E1 -15721.279,E2 -15721.279} C_VEL
LIN {X 0,Y 312.587,Z 281.173,A -85,B 0,C 180,E1 -15724.711,E2 -15724.711} C_VEL
LIN {X 0,Y 312.538,Z 281.177,A -85,B 0,C 180,E1 -15728.913,E2 -15728.913} C_VEL
LIN {X 0,Y 312.641,Z 281.164,A -85,B 0,C 180,E1 -15731.656,E2 -15731.656} C_VEL
LIN {X 0,Y 312.697,Z 281.157,A -85,B 0,C 180,E1 -15735.686,E2 -15735.686} C_VEL
LIN {X 0,Y 312.701,Z 281.157,A -85,B 0,C 180,E1 -15739.642,E2 -15739.642} C_VEL
LIN {X 0,Y 312.799,Z 281.147,A -85,B 0,C 180,E1 -15742.252,E2 -15742.252} C_VEL
LIN {X 0,Y 312.699,Z 281.156,A -85,B 0,C 180,E1 -15744.842,E2 -15744.842} C_VEL
LIN {X 0,Y 312.99,Z 281.12,A -85,B 0,C 180,E1 -15748.713,E2 -15748.713} C_VEL
LIN {X 0,Y 312.987,Z 281.12,A -85,B 0,C 180,E1 -15751.287,E2 -15751.287} C_VEL
LIN {X 0,Y 312.686,Z 281.163,A -85,B 0,C 180,E1 -15753.866,E2 -15753.866} C_VEL
LIN {X 0,Y 312.853,Z 281.137,A -85,B 0,C 180,E1 -15756.449,E2 -15756.449} C_VEL
LIN {X 0,Y 312.754,Z 281.149,A -85,B 0,C 180,E1 -15759.05,E2 -15759.05} C_VEL
LIN {X 0,Y 312.637,Z 281.164,A -85,B 0,C 180,E1 -15762.991,E2 -15762.991} C_VEL
LIN {X 0,Y 312.642,Z 281.168,A -85,B 0,C 180,E1 -15765.65,E2 -15765.65} C_VEL
LIN {X 0,Y 312.634,Z 281.166,A -85,B 0,C 180,E1 -15769.237,E2 -15769.237} C_VEL
LIN {X 0,Y 312.549,Z 281.175,A -85,B 0,C 180,E1 -15772.789,E2 -15772.789} C_VEL
LIN {X 0,Y 312.6,Z 281.169,A -85,B 0,C 180,E1 -15775.933,E2 -15775.933} C_VEL
LIN {X 0,Y 312.541,Z 281.178,A -85,B 0,C 180,E1 -15779.651,E2 -15779.651} C_VEL
LIN {X 0,Y 312.522,Z 281.179,A -85,B 0,C 180,E1 -15783.689,E2 -15783.689} C_VEL
LIN {X 0,Y 312.517,Z 281.182,A -85,B 0,C 180,E1 -15787.387,E2 -15787.387} C_VEL
LIN {X 0,Y 312.443,Z 281.19,A -85,B 0,C 180,E1 -15790.717,E2 -15790.717} C_VEL
LIN {X 0,Y 312.453,Z 281.187,A -85,B 0,C 180,E1 -15794.21,E2 -15794.21} C_VEL
LIN {X 0,Y 312.487,Z 281.182,A -85,B 0,C 180,E1 -15797.919,E2 -15797.919} C_VEL
LIN {X 0,Y 312.502,Z 281.185,A -85,B 0,C 180,E1 -15800.971,E2 -15800.971} C_VEL
LIN {X 0,Y 312.536,Z 281.177,A -85,B 0,C 180,E1 -15804.22,E2 -15804.22} C_VEL
LIN {X 0,Y 312.507,Z 281.18,A -85,B 0,C 180,E1 -15807.334,E2 -15807.334} C_VEL
LIN {X 0,Y 312.548,Z 281.175,A -85,B 0,C 180,E1 -15811.279,E2 -15811.279} C_VEL
LIN {X 0,Y 312.588,Z 281.174,A -85,B 0,C 180,E1 -15814.711,E2 -15814.711} C_VEL
LIN {X 0,Y 312.541,Z 281.177,A -85,B 0,C 180,E1 -15818.913,E2 -15818.913} C_VEL
LIN {X 0,Y 312.642,Z 281.163,A -85,B 0,C 180,E1 -15821.656,E2 -15821.656} C_VEL
LIN {X 0,Y 312.698,Z 281.156,A -85,B 0,C 180,E1 -15825.686,E2 -15825.686} C_VEL
LIN {X 0,Y 312.69,Z 281.158,A -85,B 0,C 180,E1 -15829.641,E2 -15829.641} C_VEL
LIN {X 0,Y 312.715,Z 281.152,A -85,B 0,C 180,E1 -15830.517,E2 -15830.517} C_VEL
LIN {X 0,Y 312.43,Z 281.19,A -85,B 0,C 180,E1 -15831.237,E2 -15831.237} C_VEL
LIN {X 0,Y 310.459,Z 281.442,A -85,B 0,C 180,E1 -15832.647,E2 -15832.647} C_VEL
LIN {X 0,Y 306.677,Z 281.917,A -85,B 0,C 180,E1 -15834.76,E2 -15834.76} C_VEL
LIN {X 0,Y 305.696,Z 282.034,A -85,B 0,C 180,E1 -15835.86,E2 -15835.86} C_VEL
LIN {X 0,Y 305.66,Z 282.036,A -85,B 0,C 180,E1 -15836.233,E2 -15836.233} C_VEL
LIN {X 0,Y 305.957,Z 281.996,A -85,B 0,C 180,E1 -15838.683,E2 -15838.683} C_VEL
LIN {X 0,Y 305.955,Z 281.996,A -85,B 0,C 180,E1 -15841.316,E2 -15841.316} C_VEL
LIN {X 0,Y 305.675,Z 282.032,A -85,B 0,C 180,E1 -15845.276,E2 -15845.276} C_VEL
LIN {X 0,Y 305.75,Z 282.026,A -85,B 0,C 180,E1 -15847.927,E2 -15847.927} C_VEL
LIN {X 0,Y 305.602,Z 282.044,A -85,B 0,C 180,E1 -15851.945,E2 -15851.945} C_VEL
LIN {X 0,Y 305.641,Z 282.036,A -85,B 0,C 180,E1 -15855.035,E2 -15855.035} C_VEL
LIN {X 0,Y 305.58,Z 282.046,A -85,B 0,C 180,E1 -15859.445,E2 -15859.445} C_VEL
LIN {X 0,Y 305.488,Z 282.056,A -85,B 0,C 180,E1 -15863.039,E2 -15863.039} C_VEL
LIN {X 0,Y 305.471,Z 282.061,A -85,B 0,C 180,E1 -15866.197,E2 -15866.197} C_VEL
LIN {X 0,Y 305.509,Z 282.181,A -85,B 0,C 180,E1 -15870.026,E2 -15870.026} C_VEL
LIN {X 0,Y 306.292,Z 286.925,A -85,B 0,C 180,E1 -15874.306,E2 -15874.306} C_VEL
LIN {X 0,Y 307.072,Z 291.498,A -85,B 0,C 180,E1 -15878.166,E2 -15878.166} C_VEL
LIN {X 0,Y 308.1,Z 296.68,A -85,B 0,C 180,E1 -15882.292,E2 -15882.292} C_VEL
LIN {X 0,Y 308.886,Z 301.422,A -85,B 0,C 180,E1 -15885.84,E2 -15885.84} C_VEL
LIN {X 0,Y 309.013,Z 304.281,A -85,B 0,C 180,E1 -15887.862,E2 -15887.862} C_VEL
LIN {X 0,Y 308.463,Z 308.607,A -85,B 0,C 180,E1 -15890.773,E2 -15890.773} C_VEL
LIN {X 0,Y 307.555,Z 314.12,A -85,B 0,C 180,E1 -15894.359,E2 -15894.359} C_VEL
LIN {X 0,Y 307.002,Z 318.578,A -85,B 0,C 180,E1 -15897.073,E2 -15897.073} C_VEL
LIN {X 0,Y 311.322,Z 336.881,A -85,B 0,C 180,E1 -15898.334,E2 -15898.334} C_VEL
LIN {X 0,Y 314.88,Z 353.282,A -85,B 0,C 180,E1 -15899.709,E2 -15899.709} C_VEL
LIN {X 0,Y 317.728,Z 368.536,A -85,B 0,C 180,E1 -15901.198,E2 -15901.198} C_VEL
LIN {X 0,Y 318.963,Z 376.712,A -85,B 0,C 180,E1 -15902.082,E2 -15902.082} C_VEL
LIN {X 0,Y 317.328,Z 387.392,A -85,B 0,C 180,E1 -15903.176,E2 -15903.176} C_VEL
LIN {X 0,Y 314.916,Z 400.287,A -85,B 0,C 180,E1 -15904.734,E2 -15904.734} C_VEL
LIN {X 0,Y 312.693,Z 412.299,A -85,B 0,C 180,E1 -15906.488,E2 -15906.488} C_VEL
LIN {X 0,Y 310.422,Z 424.015,A -85,B 0,C 180,E1 -15908.535,E2 -15908.535} C_VEL
LIN {X 0,Y 308.501,Z 434.354,A -85,B 0,C 180,E1 -15910.711,E2 -15910.711} C_VEL
LIN {X 0,Y 306.835,Z 443.485,A -85,B 0,C 180,E1 -15913.02,E2 -15913.02} C_VEL
LIN {X 0,Y 305.56,Z 451.104,A -85,B 0,C 180,E1 -15915.344,E2 -15915.344} C_VEL
LIN {X 0,Y 304.639,Z 458.229,A -85,B 0,C 180,E1 -15918.016,E2 -15918.016} C_VEL
LIN {X 0,Y 304.066,Z 463.809,A -85,B 0,C 180,E1 -15920.689,E2 -15920.689} C_VEL
LIN {X 0,Y 303.819,Z 467.986,A -85,B 0,C 180,E1 -15923.358,E2 -15923.358} C_VEL
LIN {X 0,Y 303.748,Z 470.841,A -85,B 0,C 180,E1 -15926.02,E2 -15926.02} C_VEL
LIN {X 0,Y 303.78,Z 472.43,A -85,B 0,C 180,E1 -15928.674,E2 -15928.674} C_VEL
LIN {X 0,Y 303.822,Z 472.767,A -85,B 0,C 180,E1 -15930,E2 -15930} C_VEL
LIN {X 0,Y 303.692,Z 472.482,A -85,B 0,C 180,E1 -15932.653,E2 -15932.653} C_VEL
LIN {X 0,Y 303.708,Z 470.97,A -85,B 0,C 180,E1 -15935.311,E2 -15935.311} C_VEL
LIN {X 0,Y 303.839,Z 468.28,A -85,B 0,C 180,E1 -15937.978,E2 -15937.978} C_VEL
LIN {X 0,Y 304.252,Z 464.41,A -85,B 0,C 180,E1 -15940.649,E2 -15940.649} C_VEL
LIN {X 0,Y 305.149,Z 459.329,A -85,B 0,C 180,E1 -15943.316,E2 -15943.316} C_VEL
LIN {X 0,Y 306.473,Z 452.95,A -85,B 0,C 180,E1 -15945.973,E2 -15945.973} C_VEL
LIN {X 0,Y 308.655,Z 444.127,A -85,B 0,C 180,E1 -15948.934,E2 -15948.934} C_VEL
LIN {X 0,Y 311.211,Z 434.738,A -85,B 0,C 180,E1 -15951.529,E2 -15951.529} C_VEL
LIN {X 0,Y 314.507,Z 423.682,A -85,B 0,C 180,E1 -15954.068,E2 -15954.068} C_VEL
LIN {X 0,Y 318.575,Z 410.705,A -85,B 0,C 180,E1 -15956.534,E2 -15956.534} C_VEL
LIN {X 0,Y 323.133,Z 396.523,A -85,B 0,C 180,E1 -15958.765,E2 -15958.765} C_VEL
LIN {X 0,Y 327.181,Z 383.874,A -85,B 0,C 180,E1 -15960.42,E2 -15960.42} C_VEL
LIN {X 0,Y 329.061,Z 366.953,A -85,B 0,C 180,E1 -15963.009,E2 -15963.009} C_VEL
LIN {X 0,Y 329.077,Z 357.931,A -85,B 0,C 180,E1 -15964.603,E2 -15964.603} C_VEL
LIN {X 0,Y 328.67,Z 350.797,A -85,B 0,C 180,E1 -15966.071,E2 -15966.071} C_VEL
LIN {X 0,Y 327.861,Z 343.142,A -85,B 0,C 180,E1 -15968.017,E2 -15968.017} C_VEL
LIN {X 0,Y 327.306,Z 336.669,A -85,B 0,C 180,E1 -15970.104,E2 -15970.104} C_VEL
LIN {X 0,Y 326.951,Z 332.175,A -85,B 0,C 180,E1 -15972.544,E2 -15972.544} C_VEL
LIN {X 0,Y 327.14,Z 330.902,A -85,B 0,C 180,E1 -15973.43,E2 -15973.43} C_VEL
LIN {X 0,Y 327.496,Z 329.991,A -85,B 0,C 180,E1 -15975.087,E2 -15975.087} C_VEL
LIN {X 0,Y 328.169,Z 330.321,A -85,B 0,C 180,E1 -15976.741,E2 -15976.741} C_VEL
LIN {X 0,Y 329.478,Z 331.908,A -85,B 0,C 180,E1 -15978.605,E2 -15978.605} C_VEL
LIN {X 0,Y 330.648,Z 333.847,A -85,B 0,C 180,E1 -15979.924,E2 -15979.924} C_VEL
LIN {X 0,Y 332.601,Z 338.269,A -85,B 0,C 180,E1 -15981.884,E2 -15981.884} C_VEL
LIN {X 0,Y 334.351,Z 343.426,A -85,B 0,C 180,E1 -15983.552,E2 -15983.552} C_VEL
LIN {X 0,Y 335.18,Z 347.047,A -85,B 0,C 180,E1 -15984.503,E2 -15984.503} C_VEL
LIN {X 0,Y 334.969,Z 348.698,A -85,B 0,C 180,E1 -15984.758,E2 -15984.758} C_VEL
LIN {X 0,Y 330.168,Z 363.818,A -85,B 0,C 180,E1 -15986.585,E2 -15986.585} C_VEL
LIN {X 0,Y 325.277,Z 378.542,A -85,B 0,C 180,E1 -15988.765,E2 -15988.765} C_VEL
LIN {X 0,Y 320.708,Z 391.704,A -85,B 0,C 180,E1 -15991.177,E2 -15991.177} C_VEL
LIN {X 0,Y 316.822,Z 402.777,A -85,B 0,C 180,E1 -15993.663,E2 -15993.663} C_VEL
LIN {X 0,Y 313.544,Z 411.939,A -85,B 0,C 180,E1 -15996.205,E2 -15996.205} C_VEL
LIN {X 0,Y 310.775,Z 419.473,A -85,B 0,C 180,E1 -15998.788,E2 -15998.788} C_VEL
LIN {X 0,Y 308.692,Z 425.543,A -85,B 0,C 180,E1 -16001.414,E2 -16001.414} C_VEL
LIN {X 0,Y 306.919,Z 430.308,A -85,B 0,C 180,E1 -16004.101,E2 -16004.101} C_VEL
LIN {X 0,Y 305.67,Z 433.633,A -85,B 0,C 180,E1 -16006.708,E2 -16006.708} C_VEL
LIN {X 0,Y 304.822,Z 435.774,A -85,B 0,C 180,E1 -16009.371,E2 -16009.371} C_VEL
LIN {X 0,Y 304.308,Z 436.673,A -85,B 0,C 180,E1 -16012.035,E2 -16012.035} C_VEL
LIN {X 0,Y 304.085,Z 436.35,A -85,B 0,C 180,E1 -16014.696,E2 -16014.696} C_VEL
LIN {X 0,Y 303.947,Z 434.817,A -85,B 0,C 180,E1 -16017.35,E2 -16017.35} C_VEL
LIN {X 0,Y 303.965,Z 432.04,A -85,B 0,C 180,E1 -16020,E2 -16020} C_VEL
LIN {X 0,Y 304.162,Z 427.973,A -85,B 0,C 180,E1 -16022.649,E2 -16022.649} C_VEL
LIN {X 0,Y 304.587,Z 424.043,A -85,B 0,C 180,E1 -16024.632,E2 -16024.632} C_VEL
LIN {X 0,Y 305.209,Z 417.481,A -85,B 0,C 180,E1 -16027.276,E2 -16027.276} C_VEL
LIN {X 0,Y 306.057,Z 409.275,A -85,B 0,C 180,E1 -16029.917,E2 -16029.917} C_VEL
LIN {X 0,Y 307.26,Z 400.573,A -85,B 0,C 180,E1 -16032.215,E2 -16032.215} C_VEL
LIN {X 0,Y 308.704,Z 390.179,A -85,B 0,C 180,E1 -16034.503,E2 -16034.503} C_VEL
LIN {X 0,Y 310.218,Z 379.682,A -85,B 0,C 180,E1 -16036.451,E2 -16036.451} C_VEL
LIN {X 0,Y 311.959,Z 367.292,A -85,B 0,C 180,E1 -16038.385,E2 -16038.385} C_VEL
LIN {X 0,Y 313.704,Z 353.756,A -85,B 0,C 180,E1 -16040.149,E2 -16040.149} C_VEL
LIN {X 0,Y 315.653,Z 338.925,A -85,B 0,C 180,E1 -16041.726,E2 -16041.726} C_VEL
LIN {X 0,Y 316.936,Z 327.074,A -85,B 0,C 180,E1 -16042.783,E2 -16042.783} C_VEL
LIN {X 0,Y 313.754,Z 313.63,A -85,B 0,C 180,E1 -16044.069,E2 -16044.069} C_VEL
LIN {X 0,Y 309.182,Z 297.291,A -85,B 0,C 180,E1 -16045.422,E2 -16045.422} C_VEL
LIN {X 0,Y 304.577,Z 282.174,A -85,B 0,C 180,E1 -16046.496,E2 -16046.496} C_VEL
LIN {X 0,Y 305,Z 282.115,A -85,B 0,C 180,E1 -16050.46,E2 -16050.46} C_VEL
LIN {X 0,Y 305.327,Z 282.074,A -85,B 0,C 180,E1 -16054.04,E2 -16054.04} C_VEL
LIN {X 0,Y 305.44,Z 282.063,A -85,B 0,C 180,E1 -16056.745,E2 -16056.745} C_VEL
LIN {X 0,Y 305.457,Z 282.061,A -85,B 0,C 180,E1 -16060.6,E2 -16060.6} C_VEL
LIN {X 0,Y 305.428,Z 282.063,A -85,B 0,C 180,E1 -16063.655,E2 -16063.655} C_VEL
LIN {X 0,Y 305.458,Z 282.059,A -85,B 0,C 180,E1 -16067.414,E2 -16067.414} C_VEL
LIN {X 0,Y 305.47,Z 282.057,A -85,B 0,C 180,E1 -16071.596,E2 -16071.596} C_VEL
LIN {X 0,Y 305.465,Z 282.061,A -85,B 0,C 180,E1 -16074.887,E2 -16074.887} C_VEL
LIN {X 0,Y 305.452,Z 282.061,A -85,B 0,C 180,E1 -16078.356,E2 -16078.356} C_VEL
LIN {X 0,Y 305.516,Z 282.052,A -85,B 0,C 180,E1 -16081.113,E2 -16081.113} C_VEL
LIN {X 0,Y 305.568,Z 282.046,A -85,B 0,C 180,E1 -16084.087,E2 -16084.087} C_VEL
LIN {X 0,Y 305.475,Z 282.061,A -85,B 0,C 180,E1 -16088.401,E2 -16088.401} C_VEL
LIN {X 0,Y 305.582,Z 282.043,A -85,B 0,C 180,E1 -16091.217,E2 -16091.217} C_VEL
LIN {X 0,Y 305.652,Z 282.033,A -85,B 0,C 180,E1 -16095.349,E2 -16095.349} C_VEL
LIN {X 0,Y 305.638,Z 282.036,A -85,B 0,C 180,E1 -16099.4,E2 -16099.4} C_VEL
LIN {X 0,Y 305.75,Z 282.026,A -85,B 0,C 180,E1 -16102.073,E2 -16102.073} C_VEL
LIN {X 0,Y 305.668,Z 282.032,A -85,B 0,C 180,E1 -16104.723,E2 -16104.723} C_VEL
LIN {X 0,Y 305.957,Z 281.996,A -85,B 0,C 180,E1 -16108.684,E2 -16108.684} C_VEL
LIN {X 0,Y 305.955,Z 281.996,A -85,B 0,C 180,E1 -16111.316,E2 -16111.316} C_VEL
LIN {X 0,Y 305.674,Z 282.032,A -85,B 0,C 180,E1 -16115.277,E2 -16115.277} C_VEL
LIN {X 0,Y 305.764,Z 282.023,A -85,B 0,C 180,E1 -16117.927,E2 -16117.927} C_VEL
LIN {X 0,Y 305.602,Z 282.043,A -85,B 0,C 180,E1 -16121.945,E2 -16121.945} C_VEL
LIN {X 0,Y 305.641,Z 282.036,A -85,B 0,C 180,E1 -16125.035,E2 -16125.035} C_VEL
LIN {X 0,Y 305.58,Z 282.047,A -85,B 0,C 180,E1 -16129.445,E2 -16129.445} C_VEL
LIN {X 0,Y 305.494,Z 282.055,A -85,B 0,C 180,E1 -16133.042,E2 -16133.042} C_VEL
LIN {X 0,Y 305.529,Z 282.049,A -85,B 0,C 180,E1 -16136.219,E2 -16136.219} C_VEL
LIN {X 0,Y 305.492,Z 282.057,A -85,B 0,C 180,E1 -16139.047,E2 -16139.047} C_VEL
LIN {X 0,Y 305.445,Z 282.06,A -85,B 0,C 180,E1 -16141.952,E2 -16141.952} C_VEL
LIN {X 0,Y 305.465,Z 282.061,A -85,B 0,C 180,E1 -16145.113,E2 -16145.113} C_VEL
LIN {X 0,Y 305.436,Z 282.062,A -85,B 0,C 180,E1 -16148.525,E2 -16148.525} C_VEL
LIN {X 0,Y 305.438,Z 282.062,A -85,B 0,C 180,E1 -16152.582,E2 -16152.582} C_VEL
LIN {X 0,Y 305.428,Z 282.062,A -85,B 0,C 180,E1 -16156.345,E2 -16156.345} C_VEL
LIN {X 0,Y 305.461,Z 282.057,A -85,B 0,C 180,E1 -16159.892,E2 -16159.892} C_VEL
LIN {X 0,Y 305.484,Z 282.055,A -85,B 0,C 180,E1 -16163.632,E2 -16163.632} C_VEL
LIN {X 0,Y 305.469,Z 282.06,A -85,B 0,C 180,E1 -16166.483,E2 -16166.483} C_VEL
LIN {X 0,Y 305.461,Z 282.057,A -85,B 0,C 180,E1 -16169.59,E2 -16169.59} C_VEL
LIN {X 0,Y 305.518,Z 282.056,A -85,B 0,C 180,E1 -16172.608,E2 -16172.608} C_VEL
LIN {X 0,Y 305.508,Z 282.051,A -85,B 0,C 180,E1 -16175.538,E2 -16175.538} C_VEL
LIN {X 0,Y 305.515,Z 282.051,A -85,B 0,C 180,E1 -16179.814,E2 -16179.814} C_VEL
LIN {X 0,Y 305.578,Z 282.046,A -85,B 0,C 180,E1 -16182.603,E2 -16182.603} C_VEL
LIN {X 0,Y 305.653,Z 282.033,A -85,B 0,C 180,E1 -16185.349,E2 -16185.349} C_VEL
LIN {X 0,Y 305.628,Z 282.037,A -85,B 0,C 180,E1 -16189.399,E2 -16189.399} C_VEL
LIN {X 0,Y 305.75,Z 282.026,A -85,B 0,C 180,E1 -16192.072,E2 -16192.072} C_VEL
LIN {X 0,Y 305.67,Z 282.032,A -85,B 0,C 180,E1 -16194.723,E2 -16194.723} C_VEL
LIN {X 0,Y 305.66,Z 282.036,A -85,B 0,C 180,E1 -16196.233,E2 -16196.233} C_VEL
LIN {X 0,Y 305.134,Z 282.1,A -85,B 0,C 180,E1 -16197.335,E2 -16197.335} C_VEL
LIN {X 0,Y 302.415,Z 282.437,A -85,B 0,C 180,E1 -16199.134,E2 -16199.134} C_VEL
LIN {X 0,Y 300.016,Z 282.736,A -85,B 0,C 180,E1 -16200.593,E2 -16200.593} C_VEL
LIN {X 0,Y 298.954,Z 282.871,A -85,B 0,C 180,E1 -16201.721,E2 -16201.721} C_VEL
LIN {X 0,Y 298.854,Z 282.878,A -85,B 0,C 180,E1 -16202.103,E2 -16202.103} C_VEL
LIN {X 0,Y 298.74,Z 282.895,A -85,B 0,C 180,E1 -16206.755,E2 -16206.755} C_VEL
LIN {X 0,Y 298.629,Z 282.911,A -85,B 0,C 180,E1 -16209.482,E2 -16209.482} C_VEL
LIN {X 0,Y 298.555,Z 282.922,A -85,B 0,C 180,E1 -16213.615,E2 -16213.615} C_VEL
LIN {X 0,Y 298.552,Z 282.918,A -85,B 0,C 180,E1 -16216.408,E2 -16216.408} C_VEL
LIN {X 0,Y 298.514,Z 282.928,A -85,B 0,C 180,E1 -16219.655,E2 -16219.655} C_VEL
LIN {X 0,Y 298.426,Z 282.939,A -85,B 0,C 180,E1 -16223.6,E2 -16223.6} C_VEL
LIN {X 0,Y 298.409,Z 282.94,A -85,B 0,C 180,E1 -16226.582,E2 -16226.582} C_VEL
LIN {X 0,Y 298.462,Z 283.107,A -85,B 0,C 180,E1 -16229.636,E2 -16229.636} C_VEL
LIN {X 0,Y 298.979,Z 286.446,A -85,B 0,C 180,E1 -16232.728,E2 -16232.728} C_VEL
LIN {X 0,Y 299.586,Z 290.04,A -85,B 0,C 180,E1 -16235.907,E2 -16235.907} C_VEL
LIN {X 0,Y 300.399,Z 294.263,A -85,B 0,C 180,E1 -16239.461,E2 -16239.461} C_VEL
LIN {X 0,Y 301.174,Z 298.166,A -85,B 0,C 180,E1 -16242.588,E2 -16242.588} C_VEL
LIN {X 0,Y 301.91,Z 302.909,A -85,B 0,C 180,E1 -16246.189,E2 -16246.189} C_VEL
LIN {X 0,Y 301.942,Z 305.633,A -85,B 0,C 180,E1 -16248.144,E2 -16248.144} C_VEL
LIN {X 0,Y 301.135,Z 310.992,A -85,B 0,C 180,E1 -16251.796,E2 -16251.796} C_VEL
LIN {X 0,Y 300.135,Z 317.073,A -85,B 0,C 180,E1 -16255.806,E2 -16255.806} C_VEL
LIN {X 0,Y 300.016,Z 318.054,A -85,B 0,C 180,E1 -16256.441,E2 -16256.441} C_VEL
LIN {X 0,Y 303.849,Z 334.293,A -85,B 0,C 180,E1 -16257.592,E2 -16257.592} C_VEL
LIN {X 0,Y 307.325,Z 350.428,A -85,B 0,C 180,E1 -16258.943,E2 -16258.943} C_VEL
LIN {X 0,Y 310.256,Z 365.482,A -85,B 0,C 180,E1 -16260.415,E2 -16260.415} C_VEL
LIN {X 0,Y 312.112,Z 377.801,A -85,B 0,C 180,E1 -16261.779,E2 -16261.779} C_VEL
LIN {X 0,Y 309.813,Z 390.921,A -85,B 0,C 180,E1 -16263.201,E2 -16263.201} C_VEL
LIN {X 0,Y 307.29,Z 404.325,A -85,B 0,C 180,E1 -16264.969,E2 -16264.969} C_VEL
LIN {X 0,Y 304.92,Z 416.607,A -85,B 0,C 180,E1 -16266.932,E2 -16266.932} C_VEL
LIN {X 0,Y 302.873,Z 427.014,A -85,B 0,C 180,E1 -16268.92,E2 -16268.92} C_VEL
LIN {X 0,Y 300.864,Z 437.266,A -85,B 0,C 180,E1 -16271.265,E2 -16271.265} C_VEL
LIN {X 0,Y 299.359,Z 445.855,A -85,B 0,C 180,E1 -16273.637,E2 -16273.637} C_VEL
LIN {X 0,Y 298.061,Z 453.917,A -85,B 0,C 180,E1 -16276.362,E2 -16276.362} C_VEL
LIN {X 0,Y 297.247,Z 460.348,A -85,B 0,C 180,E1 -16279.097,E2 -16279.097} C_VEL
LIN {X 0,Y 296.875,Z 465.318,A -85,B 0,C 180,E1 -16281.834,E2 -16281.834} C_VEL
LIN {X 0,Y 296.721,Z 468.919,A -85,B 0,C 180,E1 -16284.563,E2 -16284.563} C_VEL
LIN {X 0,Y 296.615,Z 471.221,A -85,B 0,C 180,E1 -16287.284,E2 -16287.284} C_VEL
LIN {X 0,Y 296.738,Z 472.274,A -85,B 0,C 180,E1 -16290,E2 -16290} C_VEL
LIN {X 0,Y 296.615,Z 472.043,A -85,B 0,C 180,E1 -16292.716,E2 -16292.716} C_VEL
LIN {X 0,Y 296.7,Z 470.353,A -85,B 0,C 180,E1 -16295.813,E2 -16295.813} C_VEL
LIN {X 0,Y 296.781,Z 468.037,A -85,B 0,C 180,E1 -16298.169,E2 -16298.169} C_VEL
LIN {X 0,Y 297.208,Z 464.29,A -85,B 0,C 180,E1 -16300.905,E2 -16300.905} C_VEL
LIN {X 0,Y 298.161,Z 459.317,A -85,B 0,C 180,E1 -16303.634,E2 -16303.634} C_VEL
LIN {X 0,Y 299.606,Z 453.074,A -85,B 0,C 180,E1 -16306.349,E2 -16306.349} C_VEL
LIN {X 0,Y 301.926,Z 444.51,A -85,B 0,C 180,E1 -16309.372,E2 -16309.372} C_VEL
LIN {X 0,Y 305.01,Z 434.151,A -85,B 0,C 180,E1 -16312.346,E2 -16312.346} C_VEL
LIN {X 0,Y 308.62,Z 423.224,A -85,B 0,C 180,E1 -16314.916,E2 -16314.916} C_VEL
LIN {X 0,Y 312.377,Z 412.211,A -85,B 0,C 180,E1 -16317.103,E2 -16317.103} C_VEL
LIN {X 0,Y 317.473,Z 397.592,A -85,B 0,C 180,E1 -16319.509,E2 -16319.509} C_VEL
LIN {X 0,Y 321.434,Z 386.495,A -85,B 0,C 180,E1 -16321.032,E2 -16321.032} C_VEL
LIN {X 0,Y 323.927,Z 370.154,A -85,B 0,C 180,E1 -16323.659,E2 -16323.659} C_VEL
LIN {X 0,Y 324.306,Z 362,A -85,B 0,C 180,E1 -16325.187,E2 -16325.187} C_VEL
LIN {X 0,Y 324.211,Z 354.369,A -85,B 0,C 180,E1 -16326.875,E2 -16326.875} C_VEL
LIN {X 0,Y 323.873,Z 346.758,A -85,B 0,C 180,E1 -16328.999,E2 -16328.999} C_VEL
LIN {X 0,Y 323.771,Z 342.181,A -85,B 0,C 180,E1 -16330.632,E2 -16330.632} C_VEL
LIN {X 0,Y 323.687,Z 338.984,A -85,B 0,C 180,E1 -16332.42,E2 -16332.42} C_VEL
LIN {X 0,Y 324.132,Z 336.756,A -85,B 0,C 180,E1 -16334.314,E2 -16334.314} C_VEL
LIN {X 0,Y 324.69,Z 336.528,A -85,B 0,C 180,E1 -16336.16,E2 -16336.16} C_VEL
LIN {X 0,Y 325.73,Z 337.593,A -85,B 0,C 180,E1 -16338.021,E2 -16338.021} C_VEL
LIN {X 0,Y 327.097,Z 340.112,A -85,B 0,C 180,E1 -16339.866,E2 -16339.866} C_VEL
LIN {X 0,Y 328.616,Z 344.037,A -85,B 0,C 180,E1 -16341.669,E2 -16341.669} C_VEL
LIN {X 0,Y 330.011,Z 349.252,A -85,B 0,C 180,E1 -16343.395,E2 -16343.395} C_VEL
LIN {X 0,Y 330.154,Z 351.692,A -85,B 0,C 180,E1 -16343.99,E2 -16343.99} C_VEL
LIN {X 0,Y 324.775,Z 367.141,A -85,B 0,C 180,E1 -16345.95,E2 -16345.95} C_VEL
LIN {X 0,Y 320.255,Z 379.453,A -85,B 0,C 180,E1 -16347.848,E2 -16347.848} C_VEL
LIN {X 0,Y 315.833,Z 391.173,A -85,B 0,C 180,E1 -16350.029,E2 -16350.029} C_VEL
LIN {X 0,Y 311.64,Z 402.01,A -85,B 0,C 180,E1 -16352.464,E2 -16352.464} C_VEL
LIN {X 0,Y 308.028,Z 411.335,A -85,B 0,C 180,E1 -16355.033,E2 -16355.033} C_VEL
LIN {X 0,Y 304.922,Z 419.058,A -85,B 0,C 180,E1 -16357.648,E2 -16357.648} C_VEL
LIN {X 0,Y 302.499,Z 425.274,A -85,B 0,C 180,E1 -16360.313,E2 -16360.313} C_VEL
LIN {X 0,Y 300.555,Z 430.152,A -85,B 0,C 180,E1 -16363.005,E2 -16363.005} C_VEL
LIN {X 0,Y 299.481,Z 432.915,A -85,B 0,C 180,E1 -16365.041,E2 -16365.041} C_VEL
LIN {X 0,Y 298.245,Z 435.586,A -85,B 0,C 180,E1 -16367.756,E2 -16367.756} C_VEL
